gfCNCPoint1[20427] = {X 387.5470, Y 13.9480, Z -2.1667, A 0.000, B 0.000, C 0.000 }
gfCNCPoint1[20428] = {X 387.4498, Y 13.0232, Z -2.1667, A 0.000, B 0.000, C 0.000 }
gfCNCPoint1[20429] = {X 387.4496, Y 12.1868, Z -2.1667, A 0.000, B 0.000, C 0.000 }
gfCNCPoint1[20430] = {X 387.5362, Y 11.2718, Z -2.1667, A 0.000, B 0.000, C 0.000 }
gfCNCPoint1[20431] = {X 387.7928, Y 10.3892, Z -2.1667, A 0.000, B 0.000, C 0.000 }
gfCNCPoint1[20432] = {X 388.2375, Y 9.5281, Z -2.1667, A 0.000, B 0.000, C 0.000 }
gfCNCPoint1[20433] = {X 388.8436, Y 8.7718, Z -2.1667, A 0.000, B 0.000, C 0.000 }
gfCNCPoint1[20434] = {X 389.5872, Y 8.1503, Z -2.1667, A 0.000, B 0.000, C 0.000 }
gfCNCPoint1[20435] = {X 390.4390, Y 7.6880, Z -2.1667, A 0.000, B 0.000, C 0.000 }
gfCNCPoint1[20436] = {X 391.3653, Y 7.4030, Z -2.1667, A 0.000, B 0.000, C 0.000 }
gfCNCPoint1[20437] = {X 392.3296, Y 7.3068, Z -2.1667, A 0.000, B 0.000, C 0.000 }
gfCNCPoint1[20438] = {X 399.1118, Y 7.3068, Z -2.1667, A 0.000, B 0.000, C 0.000 }
gfCNCPoint1[20439] = {X 400.0638, Y 7.4006, Z -2.1667, A 0.000, B 0.000, C 0.000 }
gfCNCPoint1[20440] = {X 400.9793, Y 7.6783, Z -2.1667, A 0.000, B 0.000, C 0.000 }
gfCNCPoint1[20441] = {X 401.8229, Y 8.1292, Z -2.1667, A 0.000, B 0.000, C 0.000 }
gfCNCPoint1[20442] = {X 402.5624, Y 8.7361, Z -2.1667, A 0.000, B 0.000, C 0.000 }
gfCNCPoint1[20443] = {X 403.1693, Y 9.4756, Z -2.1667, A 0.000, B 0.000, C 0.000 }
gfCNCPoint1[20444] = {X 403.6203, Y 10.3193, Z -2.1667, A 0.000, B 0.000, C 0.000 }
gfCNCPoint1[20445] = {X 403.8980, Y 11.2348, Z -2.1667, A 0.000, B 0.000, C 0.000 }
gfCNCPoint1[20446] = {X 403.9918, Y 12.1868, Z -2.1667, A 0.000, B 0.000, C 0.000 }
gfCNCPoint1[20447] = {X 403.9915, Y 13.0237, Z -2.1667, A 0.000, B 0.000, C 0.000 }
gfCNCPoint1[20448] = {X 403.9016, Y 13.9115, Z -2.1667, A 0.000, B 0.000, C 0.000 }
gfCNCPoint1[20449] = {X 403.6516, Y 14.7680, Z -2.1667, A 0.000, B 0.000, C 0.000 }
gfCNCPoint1[20450] = {X 405.3653, Y 17.7437, Z -2.1667, A 0.000, B 0.000, C 0.000 }
gfCNCPoint1[20451] = {X 407.2450, Y 14.6988, Z -2.1667, A 0.000, B 0.000, C 0.000 }
gfCNCPoint1[20452] = {X 407.0143, Y 13.8732, Z -2.1667, A 0.000, B 0.000, C 0.000 }
gfCNCPoint1[20453] = {X 406.9317, Y 13.0199, Z -2.1667, A 0.000, B 0.000, C 0.000 }
gfCNCPoint1[20454] = {X 406.9315, Y 12.1868, Z -2.1667, A 0.000, B 0.000, C 0.000 }
gfCNCPoint1[20455] = {X 407.0253, Y 11.2348, Z -2.1667, A 0.000, B 0.000, C 0.000 }
gfCNCPoint1[20456] = {X 407.3030, Y 10.3193, Z -2.1667, A 0.000, B 0.000, C 0.000 }
gfCNCPoint1[20457] = {X 407.7540, Y 9.4756, Z -2.1667, A 0.000, B 0.000, C 0.000 }
gfCNCPoint1[20458] = {X 408.3609, Y 8.7361, Z -2.1667, A 0.000, B 0.000, C 0.000 }
gfCNCPoint1[20459] = {X 409.1004, Y 8.1292, Z -2.1667, A 0.000, B 0.000, C 0.000 }
gfCNCPoint1[20460] = {X 409.9440, Y 7.6783, Z -2.1667, A 0.000, B 0.000, C 0.000 }
gfCNCPoint1[20461] = {X 410.8595, Y 7.4006, Z -2.1667, A 0.000, B 0.000, C 0.000 }
gfCNCPoint1[20462] = {X 411.8115, Y 7.3068, Z -2.1667, A 0.000, B 0.000, C 0.000 }
gfCNCPoint1[20463] = {X 419.3245, Y 7.3068, Z -2.1667, A 0.000, B 0.000, C 0.000 }
gfCNCPoint1[20464] = {X 420.2888, Y 7.4030, Z -2.1667, A 0.000, B 0.000, C 0.000 }
gfCNCPoint1[20465] = {X 421.2151, Y 7.6880, Z -2.1667, A 0.000, B 0.000, C 0.000 }
gfCNCPoint1[20466] = {X 422.0669, Y 8.1503, Z -2.1667, A 0.000, B 0.000, C 0.000 }
gfCNCPoint1[20467] = {X 422.8105, Y 8.7718, Z -2.1667, A 0.000, B 0.000, C 0.000 }
gfCNCPoint1[20468] = {X 423.4166, Y 9.5281, Z -2.1667, A 0.000, B 0.000, C 0.000 }
gfCNCPoint1[20469] = {X 423.8613, Y 10.3892, Z -2.1667, A 0.000, B 0.000, C 0.000 }
gfCNCPoint1[20470] = {X 424.1179, Y 11.2718, Z -2.1667, A 0.000, B 0.000, C 0.000 }
gfCNCPoint1[20471] = {X 424.2045, Y 12.1868, Z -2.1667, A 0.000, B 0.000, C 0.000 }
gfCNCPoint1[20472] = {X 424.2045, Y 12.9779, Z -2.1667, A 0.000, B 0.000, C 0.000 }
gfCNCPoint1[20473] = {X 424.1055, Y 13.9307, Z -2.1667, A 0.000, B 0.000, C 0.000 }
gfCNCPoint1[20474] = {X 423.8248, Y 14.8465, Z -2.1667, A 0.000, B 0.000, C 0.000 }
gfCNCPoint1[20475] = {X 423.3729, Y 15.6910, Z -2.1667, A 0.000, B 0.000, C 0.000 }
gfCNCPoint1[20476] = {X 422.7668, Y 16.4327, Z -2.1667, A 0.000, B 0.000, C 0.000 }
gfCNCPoint1[20477] = {X 422.0290, Y 17.0436, Z -2.1667, A 0.000, B 0.000, C 0.000 }
gfCNCPoint1[20478] = {X 421.1874, Y 17.5009, Z -2.1667, A 0.000, B 0.000, C 0.000 }
gfCNCPoint1[20479] = {X 420.5395, Y 18.3844, Z -2.1667, A 0.000, B 0.000, C 0.000 }
gfCNCPoint1[20480] = {X 419.9503, Y 19.3080, Z -2.1667, A 0.000, B 0.000, C 0.000 }
gfCNCPoint1[20481] = {X 414.1631, Y 28.6162, Z -2.1667, A 0.000, B 0.000, C 0.000 }
gfCNCPoint1[20482] = {X 422.3159, Y 33.6850, Z -2.1667, A 0.000, B 0.000, C 0.000 }
gfCNCPoint1[20483] = {X 421.8891, Y 34.3715, Z -2.1667, A 0.000, B 0.000, C 0.000 }
gfCNCPoint1[20484] = {X 422.1457, Y 34.1014, Z -2.1667, A 0.000, B 0.000, C 0.000 }
gfCNCPoint1[20485] = {X 422.4091, Y 33.8380, Z -2.1667, A 0.000, B 0.000, C 0.000 }
gfCNCPoint1[20486] = {X 422.3623, Y 33.7616, Z -2.1667, A 0.000, B 0.000, C 0.000 }
gfCNCPoint1[20487] = {X 422.3159, Y 33.6850, Z -2.1667, A 0.000, B 0.000, C 0.000 }
gfCNCPoint1[20488] = {X 420.2777, Y 32.4178, Z -2.1667, A 0.000, B 0.000, C 0.000 }
gfCNCPoint1[20489] = {X 419.3062, Y 33.9804, Z -2.1667, A 0.000, B 0.000, C 0.000 }
gfCNCPoint1[20490] = {X 419.3065, Y 38.3391, Z -2.1667, A 0.000, B 0.000, C 0.000 }
gfCNCPoint1[20491] = {X 419.9570, Y 39.7077, Z -2.1667, A 0.000, B 0.000, C 0.000 }
gfCNCPoint1[20492] = {X 420.4329, Y 41.1464, Z -2.1667, A 0.000, B 0.000, C 0.000 }
gfCNCPoint1[20493] = {X 420.6276, Y 41.1585, Z -2.1667, A 0.000, B 0.000, C 0.000 }
gfCNCPoint1[20494] = {X 420.8222, Y 41.1728, Z -2.1667, A 0.000, B 0.000, C 0.000 }
gfCNCPoint1[20495] = {X 421.2839, Y 39.7588, Z -2.1667, A 0.000, B 0.000, C 0.000 }
gfCNCPoint1[20496] = {X 421.9160, Y 38.4123, Z -2.1667, A 0.000, B 0.000, C 0.000 }
gfCNCPoint1[20497] = {X 422.7087, Y 37.1536, Z -2.1667, A 0.000, B 0.000, C 0.000 }
gfCNCPoint1[20498] = {X 423.6502, Y 36.0020, Z -2.1667, A 0.000, B 0.000, C 0.000 }
gfCNCPoint1[20499] = {X 424.3400, Y 35.3147, Z -2.1667, A 0.000, B 0.000, C 0.000 }
gfCNCPoint1[20500] = {X 425.0829, Y 34.6852, Z -2.1667, A 0.000, B 0.000, C 0.000 }
gfCNCPoint1[20501] = {X 425.4264, Y 34.0128, Z -2.1667, A 0.000, B 0.000, C 0.000 }
gfCNCPoint1[20502] = {X 424.8791, Y 33.2419, Z -2.1667, A 0.000, B 0.000, C 0.000 }
gfCNCPoint1[20503] = {X 424.3706, Y 32.4448, Z -2.1667, A 0.000, B 0.000, C 0.000 }
gfCNCPoint1[20504] = {X 423.3899, Y 30.5981, Z -2.1667, A 0.000, B 0.000, C 0.000 }
gfCNCPoint1[20505] = {X 422.6170, Y 28.6551, Z -2.1667, A 0.000, B 0.000, C 0.000 }
gfCNCPoint1[20506] = {X 420.2777, Y 32.4178, Z -2.1667, A 0.000, B 0.000, C 0.000 }
gfCNCPoint1[20507] = {X 418.2395, Y 31.1506, Z -2.1667, A 0.000, B 0.000, C 0.000 }
gfCNCPoint1[20508] = {X 416.9061, Y 33.2953, Z -2.1667, A 0.000, B 0.000, C 0.000 }
gfCNCPoint1[20509] = {X 416.9065, Y 38.9959, Z -2.1667, A 0.000, B 0.000, C 0.000 }
gfCNCPoint1[20510] = {X 417.4880, Y 40.0490, Z -2.1667, A 0.000, B 0.000, C 0.000 }
gfCNCPoint1[20511] = {X 417.9361, Y 41.1653, Z -2.1667, A 0.000, B 0.000, C 0.000 }
gfCNCPoint1[20512] = {X 418.2441, Y 42.3282, Z -2.1667, A 0.000, B 0.000, C 0.000 }
gfCNCPoint1[20513] = {X 418.4074, Y 43.5200, Z -2.1667, A 0.000, B 0.000, C 0.000 }
gfCNCPoint1[20514] = {X 419.4886, Y 43.5200, Z -2.1667, A 0.000, B 0.000, C 0.000 }
gfCNCPoint1[20515] = {X 421.1752, Y 43.6186, Z -2.1667, A 0.000, B 0.000, C 0.000 }
gfCNCPoint1[20516] = {X 422.8389, Y 43.9129, Z -2.1667, A 0.000, B 0.000, C 0.000 }
gfCNCPoint1[20517] = {X 423.0005, Y 42.4234, Z -2.1667, A 0.000, B 0.000, C 0.000 }
gfCNCPoint1[20518] = {X 423.3900, Y 40.9766, Z -2.1667, A 0.000, B 0.000, C 0.000 }
gfCNCPoint1[20519] = {X 423.9980, Y 39.6073, Z -2.1667, A 0.000, B 0.000, C 0.000 }
gfCNCPoint1[20520] = {X 424.8102, Y 38.3482, Z -2.1667, A 0.000, B 0.000, C 0.000 }
gfCNCPoint1[20521] = {X 425.8068, Y 37.2295, Z -2.1667, A 0.000, B 0.000, C 0.000 }
gfCNCPoint1[20522] = {X 426.9642, Y 36.2780, Z -2.1667, A 0.000, B 0.000, C 0.000 }
gfCNCPoint1[20523] = {X 428.2766, Y 33.7091, Z -2.1667, A 0.000, B 0.000, C 0.000 }
gfCNCPoint1[20524] = {X 427.2128, Y 32.3915, Z -2.1667, A 0.000, B 0.000, C 0.000 }
gfCNCPoint1[20525] = {X 426.2880, Y 30.9728, Z -2.1667, A 0.000, B 0.000, C 0.000 }
gfCNCPoint1[20526] = {X 425.5119, Y 29.4677, Z -2.1667, A 0.000, B 0.000, C 0.000 }
gfCNCPoint1[20527] = {X 424.8924, Y 27.8916, Z -2.1667, A 0.000, B 0.000, C 0.000 }
gfCNCPoint1[20528] = {X 424.8106, Y 27.6414, Z -2.1667, A 0.000, B 0.000, C 0.000 }
gfCNCPoint1[20529] = {X 424.7328, Y 27.3900, Z -2.1667, A 0.000, B 0.000, C 0.000 }
gfCNCPoint1[20530] = {X 424.3001, Y 25.6524, Z -2.1667, A 0.000, B 0.000, C 0.000 }
gfCNCPoint1[20531] = {X 424.0106, Y 23.8853, Z -2.1667, A 0.000, B 0.000, C 0.000 }
gfCNCPoint1[20532] = {X 423.8662, Y 22.1005, Z -2.1667, A 0.000, B 0.000, C 0.000 }
gfCNCPoint1[20533] = {X 418.2395, Y 31.1506, Z -2.1667, A 0.000, B 0.000, C 0.000 }
gfCNCPoint1[20534] = {X 416.2013, Y 29.8834, Z -2.1667, A 0.000, B 0.000, C 0.000 }
gfCNCPoint1[20535] = {X 414.5060, Y 32.6101, Z -2.1667, A 0.000, B 0.000, C 0.000 }
gfCNCPoint1[20536] = {X 414.5066, Y 39.7473, Z -2.1667, A 0.000, B 0.000, C 0.000 }
gfCNCPoint1[20537] = {X 415.1552, Y 40.7521, Z -2.1667, A 0.000, B 0.000, C 0.000 }
gfCNCPoint1[20538] = {X 415.6336, Y 41.8482, Z -2.1667, A 0.000, B 0.000, C 0.000 }
gfCNCPoint1[20539] = {X 415.9293, Y 43.0070, Z -2.1667, A 0.000, B 0.000, C 0.000 }
gfCNCPoint1[20540] = {X 416.0347, Y 44.1983, Z -2.1667, A 0.000, B 0.000, C 0.000 }
gfCNCPoint1[20541] = {X 416.0347, Y 44.9999, Z -2.1667, A 0.000, B 0.000, C 0.000 }
gfCNCPoint1[20542] = {X 416.0201, Y 45.4609, Z -2.1667, A 0.000, B 0.000, C 0.000 }
gfCNCPoint1[20543] = {X 415.9763, Y 45.9200, Z -2.1667, A 0.000, B 0.000, C 0.000 }
gfCNCPoint1[20544] = {X 419.4886, Y 45.9200, Z -2.1667, A 0.000, B 0.000, C 0.000 }
gfCNCPoint1[20545] = {X 420.8957, Y 46.0022, Z -2.1667, A 0.000, B 0.000, C 0.000 }
gfCNCPoint1[20546] = {X 422.2836, Y 46.2478, Z -2.1667, A 0.000, B 0.000, C 0.000 }
gfCNCPoint1[20547] = {X 423.4822, Y 46.5992, Z -2.1667, A 0.000, B 0.000, C 0.000 }
gfCNCPoint1[20548] = {X 424.6380, Y 47.0725, Z -2.1667, A 0.000, B 0.000, C 0.000 }
gfCNCPoint1[20549] = {X 425.7388, Y 47.6626, Z -2.1667, A 0.000, B 0.000, C 0.000 }
gfCNCPoint1[20550] = {X 425.4600, Y 46.7984, Z -2.1667, A 0.000, B 0.000, C 0.000 }
gfCNCPoint1[20551] = {X 425.2910, Y 45.9063, Z -2.1667, A 0.000, B 0.000, C 0.000 }
gfCNCPoint1[20552] = {X 425.2344, Y 45.0000, Z -2.1667, A 0.000, B 0.000, C 0.000 }
gfCNCPoint1[20553] = {X 425.2344, Y 44.2090, Z -2.1667, A 0.000, B 0.000, C 0.000 }
gfCNCPoint1[20554] = {X 425.2353, Y 44.0976, Z -2.1667, A 0.000, B 0.000, C 0.000 }
gfCNCPoint1[20555] = {X 425.2378, Y 43.9863, Z -2.1667, A 0.000, B 0.000, C 0.000 }
gfCNCPoint1[20556] = {X 425.3770, Y 42.7748, Z -2.1667, A 0.000, B 0.000, C 0.000 }
gfCNCPoint1[20557] = {X 425.7165, Y 41.6036, Z -2.1667, A 0.000, B 0.000, C 0.000 }
gfCNCPoint1[20558] = {X 426.2468, Y 40.5054, Z -2.1667, A 0.000, B 0.000, C 0.000 }
gfCNCPoint1[20559] = {X 426.9528, Y 39.5112, Z -2.1667, A 0.000, B 0.000, C 0.000 }
gfCNCPoint1[20560] = {X 427.8150, Y 38.6488, Z -2.1667, A 0.000, B 0.000, C 0.000 }
gfCNCPoint1[20561] = {X 428.8090, Y 37.9424, Z -2.1667, A 0.000, B 0.000, C 0.000 }
gfCNCPoint1[20562] = {X 431.2071, Y 33.2482, Z -2.1667, A 0.000, B 0.000, C 0.000 }
gfCNCPoint1[20563] = {X 430.0935, Y 32.1404, Z -2.1667, A 0.000, B 0.000, C 0.000 }
gfCNCPoint1[20564] = {X 429.1082, Y 30.9169, Z -2.1667, A 0.000, B 0.000, C 0.000 }
gfCNCPoint1[20565] = {X 428.2633, Y 29.5927, Z -2.1667, A 0.000, B 0.000, C 0.000 }
gfCNCPoint1[20566] = {X 427.5689, Y 28.1837, Z -2.1667, A 0.000, B 0.000, C 0.000 }
gfCNCPoint1[20567] = {X 427.0335, Y 26.7069, Z -2.1667, A 0.000, B 0.000, C 0.000 }
gfCNCPoint1[20568] = {X 426.6495, Y 25.1622, Z -2.1667, A 0.000, B 0.000, C 0.000 }
gfCNCPoint1[20569] = {X 426.3925, Y 23.5913, Z -2.1667, A 0.000, B 0.000, C 0.000 }
gfCNCPoint1[20570] = {X 426.2643, Y 22.0048, Z -2.1667, A 0.000, B 0.000, C 0.000 }
gfCNCPoint1[20571] = {X 426.2911, Y 19.9392, Z -2.1667, A 0.000, B 0.000, C 0.000 }
gfCNCPoint1[20572] = {X 426.5359, Y 17.8880, Z -2.1667, A 0.000, B 0.000, C 0.000 }
gfCNCPoint1[20573] = {X 426.9959, Y 15.8741, Z -2.1667, A 0.000, B 0.000, C 0.000 }
gfCNCPoint1[20574] = {X 427.6134, Y 14.1183, Z -2.1667, A 0.000, B 0.000, C 0.000 }
gfCNCPoint1[20575] = {X 428.4471, Y 12.4541, Z -2.1667, A 0.000, B 0.000, C 0.000 }
gfCNCPoint1[20576] = {X 429.4837, Y 10.9082, Z -2.1667, A 0.000, B 0.000, C 0.000 }
gfCNCPoint1[20577] = {X 430.7066, Y 9.5051, Z -2.1667, A 0.000, B 0.000, C 0.000 }
gfCNCPoint1[20578] = {X 426.0925, Y 9.5051, Z -2.1667, A 0.000, B 0.000, C 0.000 }
gfCNCPoint1[20579] = {X 426.3754, Y 10.3751, Z -2.1667, A 0.000, B 0.000, C 0.000 }
gfCNCPoint1[20580] = {X 426.5470, Y 11.2738, Z -2.1667, A 0.000, B 0.000, C 0.000 }
gfCNCPoint1[20581] = {X 426.6045, Y 12.1868, Z -2.1667, A 0.000, B 0.000, C 0.000 }
gfCNCPoint1[20582] = {X 426.6045, Y 12.9858, Z -2.1667, A 0.000, B 0.000, C 0.000 }
gfCNCPoint1[20583] = {X 426.4810, Y 14.2875, Z -2.1667, A 0.000, B 0.000, C 0.000 }
gfCNCPoint1[20584] = {X 426.1288, Y 15.5467, Z -2.1667, A 0.000, B 0.000, C 0.000 }
gfCNCPoint1[20585] = {X 425.5589, Y 16.7235, Z -2.1667, A 0.000, B 0.000, C 0.000 }
gfCNCPoint1[20586] = {X 424.7895, Y 17.7807, Z -2.1667, A 0.000, B 0.000, C 0.000 }
gfCNCPoint1[20587] = {X 423.8449, Y 18.6847, Z -2.1667, A 0.000, B 0.000, C 0.000 }
gfCNCPoint1[20588] = {X 422.7549, Y 19.4070, Z -2.1667, A 0.000, B 0.000, C 0.000 }
gfCNCPoint1[20589] = {X 422.3647, Y 19.9716, Z -2.1667, A 0.000, B 0.000, C 0.000 }
gfCNCPoint1[20590] = {X 422.0017, Y 20.5540, Z -2.1667, A 0.000, B 0.000, C 0.000 }
gfCNCPoint1[20591] = {X 416.2013, Y 29.8834, Z -2.1667, A 0.000, B 0.000, C 0.000 }
gfCNCPoint1[20592] = {X 414.1631, Y 28.6162, Z -2.1667, A 0.000, B 0.000, C 0.000 }
gfCNCPoint1[20593] = {X 412.1060, Y 31.9249, Z -2.1667, A 0.000, B 0.000, C 0.000 }
gfCNCPoint1[20594] = {X 412.1067, Y 40.6523, Z -2.1667, A 0.000, B 0.000, C 0.000 }
gfCNCPoint1[20595] = {X 412.7484, Y 41.4088, Z -2.1667, A 0.000, B 0.000, C 0.000 }
gfCNCPoint1[20596] = {X 413.2283, Y 42.2769, Z -2.1667, A 0.000, B 0.000, C 0.000 }
gfCNCPoint1[20597] = {X 413.5277, Y 43.2227, Z -2.1667, A 0.000, B 0.000, C 0.000 }
gfCNCPoint1[20598] = {X 413.6347, Y 44.2089, Z -2.1667, A 0.000, B 0.000, C 0.000 }
gfCNCPoint1[20599] = {X 413.6347, Y 45.0000, Z -2.1667, A 0.000, B 0.000, C 0.000 }
gfCNCPoint1[20600] = {X 413.6249, Y 45.3090, Z -2.1667, A 0.000, B 0.000, C 0.000 }
gfCNCPoint1[20601] = {X 413.5956, Y 45.6167, Z -2.1667, A 0.000, B 0.000, C 0.000 }
gfCNCPoint1[20602] = {X 413.3652, Y 46.5992, Z -2.1667, A 0.000, B 0.000, C 0.000 }
gfCNCPoint1[20603] = {X 412.9377, Y 47.5134, Z -2.1667, A 0.000, B 0.000, C 0.000 }
gfCNCPoint1[20604] = {X 412.3313, Y 48.3200, Z -2.1667, A 0.000, B 0.000, C 0.000 }
gfCNCPoint1[20605] = {X 411.9795, Y 47.9934, Z -2.1667, A 0.000, B 0.000, C 0.000 }
gfCNCPoint1[20606] = {X 411.3003, Y 48.5889, Z -2.1667, A 0.000, B 0.000, C 0.000 }
gfCNCPoint1[20607] = {X 410.5138, Y 49.0331, Z -2.1667, A 0.000, B 0.000, C 0.000 }
gfCNCPoint1[20608] = {X 409.6532, Y 49.3073, Z -2.1667, A 0.000, B 0.000, C 0.000 }
gfCNCPoint1[20609] = {X 408.7547, Y 49.4000, Z -2.1667, A 0.000, B 0.000, C 0.000 }
gfCNCPoint1[20610] = {X 402.3112, Y 49.4000, Z -2.1667, A 0.000, B 0.000, C 0.000 }
gfCNCPoint1[20611] = {X 401.3321, Y 49.2897, Z -2.1667, A 0.000, B 0.000, C 0.000 }
gfCNCPoint1[20612] = {X 400.4021, Y 48.9643, Z -2.1667, A 0.000, B 0.000, C 0.000 }
gfCNCPoint1[20613] = {X 399.5678, Y 48.4400, Z -2.1667, A 0.000, B 0.000, C 0.000 }
gfCNCPoint1[20614] = {X 398.8711, Y 47.7433, Z -2.1667, A 0.000, B 0.000, C 0.000 }
gfCNCPoint1[20615] = {X 398.3469, Y 46.9091, Z -2.1667, A 0.000, B 0.000, C 0.000 }
gfCNCPoint1[20616] = {X 398.0215, Y 45.9791, Z -2.1667, A 0.000, B 0.000, C 0.000 }
gfCNCPoint1[20617] = {X 397.9112, Y 45.0000, Z -2.1667, A 0.000, B 0.000, C 0.000 }
gfCNCPoint1[20618] = {X 397.9116, Y 44.1518, Z -2.1667, A 0.000, B 0.000, C 0.000 }
gfCNCPoint1[20619] = {X 398.0215, Y 43.2300, Z -2.1667, A 0.000, B 0.000, C 0.000 }
gfCNCPoint1[20620] = {X 398.3223, Y 42.3519, Z -2.1667, A 0.000, B 0.000, C 0.000 }
gfCNCPoint1[20621] = {X 398.8006, Y 41.5563, Z -2.1667, A 0.000, B 0.000, C 0.000 }
gfCNCPoint1[20622] = {X 399.4352, Y 40.8789, Z -2.1667, A 0.000, B 0.000, C 0.000 }
gfCNCPoint1[20623] = {X 399.4352, Y 31.6934, Z -2.1667, A 0.000, B 0.000, C 0.000 }
gfCNCPoint1[20624] = {X 393.2514, Y 20.9402, Z -2.1667, A 0.000, B 0.000, C 0.000 }
gfCNCPoint1[20625] = {X 392.4348, Y 19.5574, Z -2.1667, A 0.000, B 0.000, C 0.000 }
gfCNCPoint1[20626] = {X 391.5867, Y 18.1938, Z -2.1667, A 0.000, B 0.000, C 0.000 }
gfCNCPoint1[20627] = {X 391.1415, Y 17.5837, Z -2.1667, A 0.000, B 0.000, C 0.000 }
gfCNCPoint1[20628] = {X 390.6238, Y 17.0339, Z -2.1667, A 0.000, B 0.000, C 0.000 }
gfCNCPoint1[20629] = {X 389.8686, Y 16.6254, Z -2.1667, A 0.000, B 0.000, C 0.000 }
gfCNCPoint1[20630] = {X 389.2071, Y 16.0780, Z -2.1667, A 0.000, B 0.000, C 0.000 }
gfCNCPoint1[20631] = {X 388.6645, Y 15.4125, Z -2.1667, A 0.000, B 0.000, C 0.000 }
gfCNCPoint1[20632] = {X 388.2615, Y 14.6544, Z -2.1667, A 0.000, B 0.000, C 0.000 }
gfCNCPoint1[20633] = {X 388.0134, Y 13.8324, Z -2.1667, A 0.000, B 0.000, C 0.000 }
gfCNCPoint1[20634] = {X 387.9296, Y 12.9779, Z -2.1667, A 0.000, B 0.000, C 0.000 }
gfCNCPoint1[20635] = {X 387.9296, Y 12.1868, Z -2.1667, A 0.000, B 0.000, C 0.000 }
gfCNCPoint1[20636] = {X 388.0399, Y 11.2077, Z -2.1667, A 0.000, B 0.000, C 0.000 }
gfCNCPoint1[20637] = {X 388.3654, Y 10.2777, Z -2.1667, A 0.000, B 0.000, C 0.000 }
gfCNCPoint1[20638] = {X 388.8896, Y 9.4435, Z -2.1667, A 0.000, B 0.000, C 0.000 }
gfCNCPoint1[20639] = {X 389.5863, Y 8.7468, Z -2.1667, A 0.000, B 0.000, C 0.000 }
gfCNCPoint1[20640] = {X 390.4205, Y 8.2226, Z -2.1667, A 0.000, B 0.000, C 0.000 }
gfCNCPoint1[20641] = {X 391.3505, Y 7.8971, Z -2.1667, A 0.000, B 0.000, C 0.000 }
gfCNCPoint1[20642] = {X 392.3296, Y 7.7868, Z -2.1667, A 0.000, B 0.000, C 0.000 }
gfCNCPoint1[20643] = {X 399.1118, Y 7.7868, Z -2.1667, A 0.000, B 0.000, C 0.000 }
gfCNCPoint1[20644] = {X 400.0909, Y 7.8971, Z -2.1667, A 0.000, B 0.000, C 0.000 }
gfCNCPoint1[20645] = {X 401.0208, Y 8.2226, Z -2.1667, A 0.000, B 0.000, C 0.000 }
gfCNCPoint1[20646] = {X 401.8551, Y 8.7468, Z -2.1667, A 0.000, B 0.000, C 0.000 }
gfCNCPoint1[20647] = {X 402.5518, Y 9.4435, Z -2.1667, A 0.000, B 0.000, C 0.000 }
gfCNCPoint1[20648] = {X 403.0760, Y 10.2777, Z -2.1667, A 0.000, B 0.000, C 0.000 }
gfCNCPoint1[20649] = {X 403.4014, Y 11.2077, Z -2.1667, A 0.000, B 0.000, C 0.000 }
gfCNCPoint1[20650] = {X 403.5118, Y 12.1868, Z -2.1667, A 0.000, B 0.000, C 0.000 }
gfCNCPoint1[20651] = {X 403.5115, Y 13.0233, Z -2.1667, A 0.000, B 0.000, C 0.000 }
gfCNCPoint1[20652] = {X 403.4070, Y 13.9326, Z -2.1667, A 0.000, B 0.000, C 0.000 }
gfCNCPoint1[20653] = {X 403.1165, Y 14.8007, Z -2.1667, A 0.000, B 0.000, C 0.000 }
gfCNCPoint1[20654] = {X 405.3510, Y 18.6806, Z -2.1667, A 0.000, B 0.000, C 0.000 }
gfCNCPoint1[20655] = {X 407.7814, Y 14.7438, Z -2.1667, A 0.000, B 0.000, C 0.000 }
gfCNCPoint1[20656] = {X 407.5050, Y 13.8800, Z -2.1667, A 0.000, B 0.000, C 0.000 }
gfCNCPoint1[20657] = {X 407.4115, Y 12.9779, Z -2.1667, A 0.000, B 0.000, C 0.000 }
gfCNCPoint1[20658] = {X 407.4115, Y 12.1868, Z -2.1667, A 0.000, B 0.000, C 0.000 }
gfCNCPoint1[20659] = {X 407.5219, Y 11.2077, Z -2.1667, A 0.000, B 0.000, C 0.000 }
gfCNCPoint1[20660] = {X 407.8473, Y 10.2777, Z -2.1667, A 0.000, B 0.000, C 0.000 }
gfCNCPoint1[20661] = {X 408.3715, Y 9.4435, Z -2.1667, A 0.000, B 0.000, C 0.000 }
gfCNCPoint1[20662] = {X 409.0682, Y 8.7468, Z -2.1667, A 0.000, B 0.000, C 0.000 }
gfCNCPoint1[20663] = {X 409.9024, Y 8.2226, Z -2.1667, A 0.000, B 0.000, C 0.000 }
gfCNCPoint1[20664] = {X 410.8324, Y 7.8971, Z -2.1667, A 0.000, B 0.000, C 0.000 }
gfCNCPoint1[20665] = {X 411.8115, Y 7.7868, Z -2.1667, A 0.000, B 0.000, C 0.000 }
gfCNCPoint1[20666] = {X 419.3245, Y 7.7868, Z -2.1667, A 0.000, B 0.000, C 0.000 }
gfCNCPoint1[20667] = {X 420.3036, Y 7.8971, Z -2.1667, A 0.000, B 0.000, C 0.000 }
gfCNCPoint1[20668] = {X 421.2335, Y 8.2226, Z -2.1667, A 0.000, B 0.000, C 0.000 }
gfCNCPoint1[20669] = {X 422.0678, Y 8.7468, Z -2.1667, A 0.000, B 0.000, C 0.000 }
gfCNCPoint1[20670] = {X 422.7645, Y 9.4435, Z -2.1667, A 0.000, B 0.000, C 0.000 }
gfCNCPoint1[20671] = {X 423.2887, Y 10.2777, Z -2.1667, A 0.000, B 0.000, C 0.000 }
gfCNCPoint1[20672] = {X 423.6141, Y 11.2077, Z -2.1667, A 0.000, B 0.000, C 0.000 }
gfCNCPoint1[20673] = {X 423.7245, Y 12.1868, Z -2.1667, A 0.000, B 0.000, C 0.000 }
gfCNCPoint1[20674] = {X 423.7244, Y 12.9811, Z -2.1667, A 0.000, B 0.000, C 0.000 }
gfCNCPoint1[20675] = {X 423.6301, Y 13.8598, Z -2.1667, A 0.000, B 0.000, C 0.000 }
gfCNCPoint1[20676] = {X 423.3645, Y 14.7028, Z -2.1667, A 0.000, B 0.000, C 0.000 }
gfCNCPoint1[20677] = {X 422.9382, Y 15.4769, Z -2.1667, A 0.000, B 0.000, C 0.000 }
gfCNCPoint1[20678] = {X 422.3679, Y 16.1520, Z -2.1667, A 0.000, B 0.000, C 0.000 }
gfCNCPoint1[20679] = {X 421.6758, Y 16.7016, Z -2.1667, A 0.000, B 0.000, C 0.000 }
gfCNCPoint1[20680] = {X 420.8891, Y 17.1042, Z -2.1667, A 0.000, B 0.000, C 0.000 }
gfCNCPoint1[20681] = {X 420.1821, Y 18.0570, Z -2.1667, A 0.000, B 0.000, C 0.000 }
gfCNCPoint1[20682] = {X 419.5419, Y 19.0558, Z -2.1667, A 0.000, B 0.000, C 0.000 }
gfCNCPoint1[20683] = {X 418.0618, Y 21.4528, Z -2.1667, A 0.000, B 0.000, C 0.000 }
gfCNCPoint1[20684] = {X 411.6260, Y 31.7877, Z -2.1667, A 0.000, B 0.000, C 0.000 }
gfCNCPoint1[20685] = {X 411.6267, Y 40.8621, Z -2.1667, A 0.000, B 0.000, C 0.000 }
gfCNCPoint1[20686] = {X 412.2657, Y 41.5589, Z -2.1667, A 0.000, B 0.000, C 0.000 }
gfCNCPoint1[20687] = {X 412.7461, Y 42.3733, Z -2.1667, A 0.000, B 0.000, C 0.000 }
gfCNCPoint1[20688] = {X 413.0467, Y 43.2696, Z -2.1667, A 0.000, B 0.000, C 0.000 }
gfCNCPoint1[20689] = {X 413.1547, Y 44.2089, Z -2.1667, A 0.000, B 0.000, C 0.000 }
gfCNCPoint1[20690] = {X 413.1545, Y 45.0423, Z -2.1667, A 0.000, B 0.000, C 0.000 }
gfCNCPoint1[20691] = {X 413.0719, Y 45.8494, Z -2.1667, A 0.000, B 0.000, C 0.000 }
gfCNCPoint1[20692] = {X 412.8426, Y 46.6276, Z -2.1667, A 0.000, B 0.000, C 0.000 }
gfCNCPoint1[20693] = {X 412.4743, Y 47.3505, Z -2.1667, A 0.000, B 0.000, C 0.000 }
gfCNCPoint1[20694] = {X 411.9795, Y 47.9934, Z -2.1667, A 0.000, B 0.000, C 0.000 }
gfCNCPoint1[20695] = {X 412.3313, Y 48.3200, Z -2.1667, A 0.000, B 0.000, C 0.000 }
gfCNCPoint1[20696] = {X 419.4886, Y 48.3200, Z -2.1667, A 0.000, B 0.000, C 0.000 }
gfCNCPoint1[20697] = {X 420.8006, Y 48.4093, Z -2.1667, A 0.000, B 0.000, C 0.000 }
gfCNCPoint1[20698] = {X 422.0883, Y 48.6756, Z -2.1667, A 0.000, B 0.000, C 0.000 }
gfCNCPoint1[20699] = {X 423.3281, Y 49.1140, Z -2.1667, A 0.000, B 0.000, C 0.000 }
gfCNCPoint1[20700] = {X 424.4970, Y 49.7164, Z -2.1667, A 0.000, B 0.000, C 0.000 }
gfCNCPoint1[20701] = {X 425.4625, Y 50.3832, Z -2.1667, A 0.000, B 0.000, C 0.000 }
gfCNCPoint1[20702] = {X 426.3402, Y 51.1620, Z -2.1667, A 0.000, B 0.000, C 0.000 }
gfCNCPoint1[20703] = {X 427.1172, Y 52.0412, Z -2.1667, A 0.000, B 0.000, C 0.000 }
gfCNCPoint1[20704] = {X 427.7821, Y 53.0080, Z -2.1667, A 0.000, B 0.000, C 0.000 }
gfCNCPoint1[20705] = {X 428.1269, Y 53.6317, Z -2.1667, A 0.000, B 0.000, C 0.000 }
gfCNCPoint1[20706] = {X 428.4249, Y 54.2792, Z -2.1667, A 0.000, B 0.000, C 0.000 }
gfCNCPoint1[20707] = {X 431.5823, Y 55.5098, Z -2.1667, A 0.000, B 0.000, C 0.000 }
gfCNCPoint1[20708] = {X 439.8770, Y 58.8007, Z -2.1667, A 0.000, B 0.000, C 0.000 }
gfCNCPoint1[20709] = {X 441.6471, Y 54.3390, Z -2.1667, A 0.000, B 0.000, C 0.000 }
gfCNCPoint1[20710] = {X 444.2222, Y 55.3606, Z -2.1667, A 0.000, B 0.000, C 0.000 }
gfCNCPoint1[20711] = {X 444.5425, Y 54.0020, Z -2.1667, A 0.000, B 0.000, C 0.000 }
gfCNCPoint1[20712] = {X 444.9921, Y 52.6806, Z -2.1667, A 0.000, B 0.000, C 0.000 }
gfCNCPoint1[20713] = {X 443.9519, Y 53.3765, Z -2.1667, A 0.000, B 0.000, C 0.000 }
gfCNCPoint1[20714] = {X 442.8307, Y 53.9324, Z -2.1667, A 0.000, B 0.000, C 0.000 }
gfCNCPoint1[20715] = {X 441.6471, Y 54.3390, Z -2.1667, A 0.000, B 0.000, C 0.000 }
gfCNCPoint1[20716] = {X 440.7621, Y 56.5698, Z -2.1667, A 0.000, B 0.000, C 0.000 }
gfCNCPoint1[20717] = {X 446.3797, Y 58.7986, Z -2.1667, A 0.000, B 0.000, C 0.000 }
gfCNCPoint1[20718] = {X 446.3796, Y 58.0000, Z -2.1667, A 0.000, B 0.000, C 0.000 }
gfCNCPoint1[20719] = {X 446.4303, Y 56.8944, Z -2.1667, A 0.000, B 0.000, C 0.000 }
gfCNCPoint1[20720] = {X 446.5820, Y 55.7981, Z -2.1667, A 0.000, B 0.000, C 0.000 }
gfCNCPoint1[20721] = {X 446.8492, Y 54.6647, Z -2.1667, A 0.000, B 0.000, C 0.000 }
gfCNCPoint1[20722] = {X 447.2243, Y 53.5622, Z -2.1667, A 0.000, B 0.000, C 0.000 }
gfCNCPoint1[20723] = {X 447.8767, Y 52.1752, Z -2.1667, A 0.000, B 0.000, C 0.000 }
gfCNCPoint1[20724] = {X 448.6995, Y 50.8820, Z -2.1667, A 0.000, B 0.000, C 0.000 }
gfCNCPoint1[20725] = {X 447.8224, Y 50.1272, Z -2.1667, A 0.000, B 0.000, C 0.000 }
gfCNCPoint1[20726] = {X 447.0760, Y 49.2431, Z -2.1667, A 0.000, B 0.000, C 0.000 }
gfCNCPoint1[20727] = {X 446.4792, Y 48.2518, Z -2.1667, A 0.000, B 0.000, C 0.000 }
gfCNCPoint1[20728] = {X 446.0469, Y 47.1785, Z -2.1667, A 0.000, B 0.000, C 0.000 }
gfCNCPoint1[20729] = {X 445.6333, Y 48.2126, Z -2.1667, A 0.000, B 0.000, C 0.000 }
gfCNCPoint1[20730] = {X 445.0668, Y 49.1715, Z -2.1667, A 0.000, B 0.000, C 0.000 }
gfCNCPoint1[20731] = {X 444.3606, Y 50.0328, Z -2.1667, A 0.000, B 0.000, C 0.000 }
gfCNCPoint1[20732] = {X 443.5314, Y 50.7763, Z -2.1667, A 0.000, B 0.000, C 0.000 }
gfCNCPoint1[20733] = {X 442.7491, Y 51.2997, Z -2.1667, A 0.000, B 0.000, C 0.000 }
gfCNCPoint1[20734] = {X 441.9059, Y 51.7177, Z -2.1667, A 0.000, B 0.000, C 0.000 }
gfCNCPoint1[20735] = {X 441.0157, Y 52.0235, Z -2.1667, A 0.000, B 0.000, C 0.000 }
gfCNCPoint1[20736] = {X 440.0666, Y 52.2156, Z -2.1667, A 0.000, B 0.000, C 0.000 }
gfCNCPoint1[20737] = {X 439.1005, Y 52.2800, Z -2.1667, A 0.000, B 0.000, C 0.000 }
gfCNCPoint1[20738] = {X 432.5144, Y 52.2800, Z -2.1667, A 0.000, B 0.000, C 0.000 }
gfCNCPoint1[20739] = {X 431.6034, Y 52.2228, Z -2.1667, A 0.000, B 0.000, C 0.000 }
gfCNCPoint1[20740] = {X 430.7066, Y 52.0520, Z -2.1667, A 0.000, B 0.000, C 0.000 }
gfCNCPoint1[20741] = {X 429.8384, Y 51.7703, Z -2.1667, A 0.000, B 0.000, C 0.000 }
gfCNCPoint1[20742] = {X 430.0172, Y 52.0776, Z -2.1667, A 0.000, B 0.000, C 0.000 }
gfCNCPoint1[20743] = {X 430.1870, Y 52.3901, Z -2.1667, A 0.000, B 0.000, C 0.000 }
gfCNCPoint1[20744] = {X 432.4640, Y 53.2776, Z -2.1667, A 0.000, B 0.000, C 0.000 }
gfCNCPoint1[20745] = {X 440.7621, Y 56.5698, Z -2.1667, A 0.000, B 0.000, C 0.000 }
gfCNCPoint1[20746] = {X 439.8770, Y 58.8007, Z -2.1667, A 0.000, B 0.000, C 0.000 }
gfCNCPoint1[20747] = {X 449.5098, Y 62.6225, Z -2.1667, A 0.000, B 0.000, C 0.000 }
gfCNCPoint1[20748] = {X 449.1115, Y 61.4473, Z -2.1667, A 0.000, B 0.000, C 0.000 }
gfCNCPoint1[20749] = {X 448.8668, Y 60.2308, Z -2.1667, A 0.000, B 0.000, C 0.000 }
gfCNCPoint1[20750] = {X 448.7798, Y 58.9930, Z -2.1667, A 0.000, B 0.000, C 0.000 }
gfCNCPoint1[20751] = {X 448.7796, Y 58.0000, Z -2.1667, A 0.000, B 0.000, C 0.000 }
gfCNCPoint1[20752] = {X 448.8564, Y 56.7833, Z -2.1667, A 0.000, B 0.000, C 0.000 }
gfCNCPoint1[20753] = {X 449.0855, Y 55.5859, Z -2.1667, A 0.000, B 0.000, C 0.000 }
gfCNCPoint1[20754] = {X 449.4632, Y 54.4268, Z -2.1667, A 0.000, B 0.000, C 0.000 }
gfCNCPoint1[20755] = {X 449.9837, Y 53.3244, Z -2.1667, A 0.000, B 0.000, C 0.000 }
gfCNCPoint1[20756] = {X 450.6386, Y 52.2961, Z -2.1667, A 0.000, B 0.000, C 0.000 }
gfCNCPoint1[20757] = {X 451.3887, Y 51.3890, Z -2.1667, A 0.000, B 0.000, C 0.000 }
gfCNCPoint1[20758] = {X 452.2434, Y 50.5796, Z -2.1667, A 0.000, B 0.000, C 0.000 }
gfCNCPoint1[20759] = {X 453.1901, Y 49.8800, Z -2.1667, A 0.000, B 0.000, C 0.000 }
gfCNCPoint1[20760] = {X 452.3731, Y 49.8442, Z -2.1667, A 0.000, B 0.000, C 0.000 }
gfCNCPoint1[20761] = {X 451.5735, Y 49.6724, Z -2.1667, A 0.000, B 0.000, C 0.000 }
gfCNCPoint1[20762] = {X 450.8138, Y 49.3696, Z -2.1667, A 0.000, B 0.000, C 0.000 }
gfCNCPoint1[20763] = {X 450.1154, Y 48.9441, Z -2.1667, A 0.000, B 0.000, C 0.000 }
gfCNCPoint1[20764] = {X 449.3503, Y 48.2496, Z -2.1667, A 0.000, B 0.000, C 0.000 }
gfCNCPoint1[20765] = {X 448.7486, Y 47.4095, Z -2.1667, A 0.000, B 0.000, C 0.000 }
gfCNCPoint1[20766] = {X 448.3373, Y 46.4616, Z -2.1667, A 0.000, B 0.000, C 0.000 }
gfCNCPoint1[20767] = {X 448.1732, Y 45.7588, Z -2.1667, A 0.000, B 0.000, C 0.000 }
gfCNCPoint1[20768] = {X 448.1146, Y 45.0395, Z -2.1667, A 0.000, B 0.000, C 0.000 }
gfCNCPoint1[20769] = {X 448.1149, Y 44.1416, Z -2.1667, A 0.000, B 0.000, C 0.000 }
gfCNCPoint1[20770] = {X 448.2252, Y 43.1751, Z -2.1667, A 0.000, B 0.000, C 0.000 }
gfCNCPoint1[20771] = {X 448.5250, Y 42.2497, Z -2.1667, A 0.000, B 0.000, C 0.000 }
gfCNCPoint1[20772] = {X 449.0024, Y 41.4020, Z -2.1667, A 0.000, B 0.000, C 0.000 }
gfCNCPoint1[20773] = {X 449.6384, Y 40.6660, Z -2.1667, A 0.000, B 0.000, C 0.000 }
gfCNCPoint1[20774] = {X 449.6384, Y 35.0338, Z -2.1667, A 0.000, B 0.000, C 0.000 }
gfCNCPoint1[20775] = {X 447.8156, Y 35.0338, Z -2.1667, A 0.000, B 0.000, C 0.000 }
gfCNCPoint1[20776] = {X 443.7924, Y 42.8669, Z -2.1667, A 0.000, B 0.000, C 0.000 }
gfCNCPoint1[20777] = {X 443.9301, Y 43.5098, Z -2.1667, A 0.000, B 0.000, C 0.000 }
gfCNCPoint1[20778] = {X 443.9803, Y 44.1653, Z -2.1667, A 0.000, B 0.000, C 0.000 }
gfCNCPoint1[20779] = {X 443.9805, Y 45.0000, Z -2.1667, A 0.000, B 0.000, C 0.000 }
gfCNCPoint1[20780] = {X 443.9242, Y 45.7387, Z -2.1667, A 0.000, B 0.000, C 0.000 }
gfCNCPoint1[20781] = {X 443.7568, Y 46.4603, Z -2.1667, A 0.000, B 0.000, C 0.000 }
gfCNCPoint1[20782] = {X 443.3474, Y 47.4038, Z -2.1667, A 0.000, B 0.000, C 0.000 }
gfCNCPoint1[20783] = {X 442.7493, Y 48.2405, Z -2.1667, A 0.000, B 0.000, C 0.000 }
gfCNCPoint1[20784] = {X 441.9891, Y 48.9332, Z -2.1667, A 0.000, B 0.000, C 0.000 }
gfCNCPoint1[20785] = {X 441.1006, Y 49.4513, Z -2.1667, A 0.000, B 0.000, C 0.000 }
gfCNCPoint1[20786] = {X 440.1232, Y 49.7716, Z -2.1667, A 0.000, B 0.000, C 0.000 }
gfCNCPoint1[20787] = {X 439.1005, Y 49.8800, Z -2.1667, A 0.000, B 0.000, C 0.000 }
gfCNCPoint1[20788] = {X 432.5144, Y 49.8800, Z -2.1667, A 0.000, B 0.000, C 0.000 }
gfCNCPoint1[20789] = {X 431.6014, Y 49.7938, Z -2.1667, A 0.000, B 0.000, C 0.000 }
gfCNCPoint1[20790] = {X 430.7206, Y 49.5383, Z -2.1667, A 0.000, B 0.000, C 0.000 }
gfCNCPoint1[20791] = {X 429.8343, Y 49.0782, Z -2.1667, A 0.000, B 0.000, C 0.000 }
gfCNCPoint1[20792] = {X 429.0603, Y 48.4473, Z -2.1667, A 0.000, B 0.000, C 0.000 }
gfCNCPoint1[20793] = {X 428.4309, Y 47.6720, Z -2.1667, A 0.000, B 0.000, C 0.000 }
gfCNCPoint1[20794] = {X 427.9725, Y 46.7848, Z -2.1667, A 0.000, B 0.000, C 0.000 }
gfCNCPoint1[20795] = {X 427.7197, Y 45.9083, Z -2.1667, A 0.000, B 0.000, C 0.000 }
gfCNCPoint1[20796] = {X 427.6344, Y 45.0000, Z -2.1667, A 0.000, B 0.000, C 0.000 }
gfCNCPoint1[20797] = {X 427.6344, Y 44.2089, Z -2.1667, A 0.000, B 0.000, C 0.000 }
gfCNCPoint1[20798] = {X 427.7263, Y 43.2661, Z -2.1667, A 0.000, B 0.000, C 0.000 }
gfCNCPoint1[20799] = {X 427.9987, Y 42.3588, Z -2.1667, A 0.000, B 0.000, C 0.000 }
gfCNCPoint1[20800] = {X 428.4411, Y 41.5213, Z -2.1667, A 0.000, B 0.000, C 0.000 }
gfCNCPoint1[20801] = {X 429.0371, Y 40.7849, Z -2.1667, A 0.000, B 0.000, C 0.000 }
gfCNCPoint1[20802] = {X 429.7641, Y 40.1776, Z -2.1667, A 0.000, B 0.000, C 0.000 }
gfCNCPoint1[20803] = {X 430.5947, Y 39.7222, Z -2.1667, A 0.000, B 0.000, C 0.000 }
gfCNCPoint1[20804] = {X 434.2535, Y 32.5606, Z -2.1667, A 0.000, B 0.000, C 0.000 }
gfCNCPoint1[20805] = {X 432.9192, Y 31.5578, Z -2.1667, A 0.000, B 0.000, C 0.000 }
gfCNCPoint1[20806] = {X 431.7387, Y 30.3780, Z -2.1667, A 0.000, B 0.000, C 0.000 }
gfCNCPoint1[20807] = {X 430.7351, Y 29.0444, Z -2.1667, A 0.000, B 0.000, C 0.000 }
gfCNCPoint1[20808] = {X 429.9283, Y 27.5833, Z -2.1667, A 0.000, B 0.000, C 0.000 }
gfCNCPoint1[20809] = {X 429.3342, Y 26.0236, Z -2.1667, A 0.000, B 0.000, C 0.000 }
gfCNCPoint1[20810] = {X 428.9002, Y 24.1500, Z -2.1667, A 0.000, B 0.000, C 0.000 }
gfCNCPoint1[20811] = {X 428.6788, Y 22.2397, Z -2.1667, A 0.000, B 0.000, C 0.000 }
gfCNCPoint1[20812] = {X 428.6728, Y 20.3166, Z -2.1667, A 0.000, B 0.000, C 0.000 }
gfCNCPoint1[20813] = {X 428.8824, Y 18.4049, Z -2.1667, A 0.000, B 0.000, C 0.000 }
gfCNCPoint1[20814] = {X 429.3049, Y 16.5287, Z -2.1667, A 0.000, B 0.000, C 0.000 }
gfCNCPoint1[20815] = {X 429.8219, Y 15.0577, Z -2.1667, A 0.000, B 0.000, C 0.000 }
gfCNCPoint1[20816] = {X 430.5201, Y 13.6636, Z -2.1667, A 0.000, B 0.000, C 0.000 }
gfCNCPoint1[20817] = {X 431.3883, Y 12.3684, Z -2.1667, A 0.000, B 0.000, C 0.000 }
gfCNCPoint1[20818] = {X 432.4128, Y 11.1930, Z -2.1667, A 0.000, B 0.000, C 0.000 }
gfCNCPoint1[20819] = {X 433.6949, Y 10.0650, Z -2.1667, A 0.000, B 0.000, C 0.000 }
gfCNCPoint1[20820] = {X 435.1203, Y 9.1245, Z -2.1667, A 0.000, B 0.000, C 0.000 }
gfCNCPoint1[20821] = {X 436.6618, Y 8.3896, Z -2.1667, A 0.000, B 0.000, C 0.000 }
gfCNCPoint1[20822] = {X 438.2899, Y 7.8744, Z -2.1667, A 0.000, B 0.000, C 0.000 }
gfCNCPoint1[20823] = {X 439.9586, Y 7.5567, Z -2.1667, A 0.000, B 0.000, C 0.000 }
gfCNCPoint1[20824] = {X 441.6470, Y 7.3700, Z -2.1667, A 0.000, B 0.000, C 0.000 }
gfCNCPoint1[20825] = {X 443.3447, Y 7.3156, Z -2.1667, A 0.000, B 0.000, C 0.000 }
gfCNCPoint1[20826] = {X 444.0315, Y 7.3116, Z -2.1667, A 0.000, B 0.000, C 0.000 }
gfCNCPoint1[20827] = {X 459.4465, Y 7.3116, Z -2.1667, A 0.000, B 0.000, C 0.000 }
gfCNCPoint1[20828] = {X 460.4093, Y 7.4076, Z -2.1667, A 0.000, B 0.000, C 0.000 }
gfCNCPoint1[20829] = {X 461.3340, Y 7.6921, Z -2.1667, A 0.000, B 0.000, C 0.000 }
gfCNCPoint1[20830] = {X 462.1843, Y 8.1537, Z -2.1667, A 0.000, B 0.000, C 0.000 }
gfCNCPoint1[20831] = {X 462.9266, Y 8.7742, Z -2.1667, A 0.000, B 0.000, C 0.000 }
gfCNCPoint1[20832] = {X 463.5317, Y 9.5293, Z -2.1667, A 0.000, B 0.000, C 0.000 }
gfCNCPoint1[20833] = {X 463.9756, Y 10.3889, Z -2.1667, A 0.000, B 0.000, C 0.000 }
gfCNCPoint1[20834] = {X 464.2316, Y 11.2698, Z -2.1667, A 0.000, B 0.000, C 0.000 }
gfCNCPoint1[20835] = {X 464.3179, Y 12.1830, Z -2.1667, A 0.000, B 0.000, C 0.000 }
gfCNCPoint1[20836] = {X 464.3177, Y 13.0247, Z -2.1667, A 0.000, B 0.000, C 0.000 }
gfCNCPoint1[20837] = {X 464.2101, Y 13.9983, Z -2.1667, A 0.000, B 0.000, C 0.000 }
gfCNCPoint1[20838] = {X 463.9102, Y 14.9307, Z -2.1667, A 0.000, B 0.000, C 0.000 }
gfCNCPoint1[20839] = {X 463.4302, Y 15.7845, Z -2.1667, A 0.000, B 0.000, C 0.000 }
gfCNCPoint1[20840] = {X 462.7893, Y 16.5252, Z -2.1667, A 0.000, B 0.000, C 0.000 }
gfCNCPoint1[20841] = {X 462.7890, Y 16.7699, Z -2.1667, A 0.000, B 0.000, C 0.000 }
gfCNCPoint1[20842] = {X 462.7894, Y 25.8689, Z -2.1667, A 0.000, B 0.000, C 0.000 }
gfCNCPoint1[20843] = {X 467.5894, Y 25.8687, Z -2.1667, A 0.000, B 0.000, C 0.000 }
gfCNCPoint1[20844] = {X 467.5900, Y 38.9891, Z -2.1667, A 0.000, B 0.000, C 0.000 }
gfCNCPoint1[20845] = {X 467.6015, Y 39.0069, Z -2.1667, A 0.000, B 0.000, C 0.000 }
gfCNCPoint1[20846] = {X 468.3506, Y 37.9855, Z -2.1667, A 0.000, B 0.000, C 0.000 }
gfCNCPoint1[20847] = {X 469.2267, Y 37.0706, Z -2.1667, A 0.000, B 0.000, C 0.000 }
gfCNCPoint1[20848] = {X 470.2148, Y 36.2780, Z -2.1667, A 0.000, B 0.000, C 0.000 }
gfCNCPoint1[20849] = {X 471.5281, Y 33.7073, Z -2.1667, A 0.000, B 0.000, C 0.000 }
gfCNCPoint1[20850] = {X 470.4813, Y 32.4114, Z -2.1667, A 0.000, B 0.000, C 0.000 }
gfCNCPoint1[20851] = {X 469.5678, Y 31.0183, Z -2.1667, A 0.000, B 0.000, C 0.000 }
gfCNCPoint1[20852] = {X 468.7965, Y 29.5417, Z -2.1667, A 0.000, B 0.000, C 0.000 }
gfCNCPoint1[20853] = {X 468.1749, Y 27.9961, Z -2.1667, A 0.000, B 0.000, C 0.000 }
gfCNCPoint1[20854] = {X 467.7092, Y 26.3966, Z -2.1667, A 0.000, B 0.000, C 0.000 }
gfCNCPoint1[20855] = {X 467.6477, Y 26.1330, Z -2.1667, A 0.000, B 0.000, C 0.000 }
gfCNCPoint1[20856] = {X 467.5894, Y 25.8687, Z -2.1667, A 0.000, B 0.000, C 0.000 }
gfCNCPoint1[20857] = {X 465.1894, Y 25.8688, Z -2.1667, A 0.000, B 0.000, C 0.000 }
gfCNCPoint1[20858] = {X 465.1901, Y 39.7466, Z -2.1667, A 0.000, B 0.000, C 0.000 }
gfCNCPoint1[20859] = {X 465.3901, Y 40.0171, Z -2.1667, A 0.000, B 0.000, C 0.000 }
gfCNCPoint1[20860] = {X 465.5774, Y 40.2966, Z -2.1667, A 0.000, B 0.000, C 0.000 }
gfCNCPoint1[20861] = {X 466.0634, Y 41.1919, Z -2.1667, A 0.000, B 0.000, C 0.000 }
gfCNCPoint1[20862] = {X 466.4196, Y 42.1462, Z -2.1667, A 0.000, B 0.000, C 0.000 }
gfCNCPoint1[20863] = {X 466.6392, Y 43.1408, Z -2.1667, A 0.000, B 0.000, C 0.000 }
gfCNCPoint1[20864] = {X 466.7178, Y 44.1564, Z -2.1667, A 0.000, B 0.000, C 0.000 }
gfCNCPoint1[20865] = {X 466.7179, Y 45.0000, Z -2.1667, A 0.000, B 0.000, C 0.000 }
gfCNCPoint1[20866] = {X 466.7033, Y 45.4609, Z -2.1667, A 0.000, B 0.000, C 0.000 }
gfCNCPoint1[20867] = {X 466.6596, Y 45.9200, Z -2.1667, A 0.000, B 0.000, C 0.000 }
gfCNCPoint1[20868] = {X 468.5433, Y 45.9200, Z -2.1667, A 0.000, B 0.000, C 0.000 }
gfCNCPoint1[20869] = {X 468.4996, Y 45.4609, Z -2.1667, A 0.000, B 0.000, C 0.000 }
gfCNCPoint1[20870] = {X 468.4850, Y 45.0000, Z -2.1667, A 0.000, B 0.000, C 0.000 }
gfCNCPoint1[20871] = {X 468.4850, Y 44.2090, Z -2.1667, A 0.000, B 0.000, C 0.000 }
gfCNCPoint1[20872] = {X 468.5580, Y 43.1798, Z -2.1667, A 0.000, B 0.000, C 0.000 }
gfCNCPoint1[20873] = {X 468.7759, Y 42.1714, Z -2.1667, A 0.000, B 0.000, C 0.000 }
gfCNCPoint1[20874] = {X 469.1341, Y 41.2038, Z -2.1667, A 0.000, B 0.000, C 0.000 }
gfCNCPoint1[20875] = {X 469.6255, Y 40.2966, Z -2.1667, A 0.000, B 0.000, C 0.000 }
gfCNCPoint1[20876] = {X 470.3102, Y 39.3876, Z -2.1667, A 0.000, B 0.000, C 0.000 }
gfCNCPoint1[20877] = {X 471.1282, Y 38.5964, Z -2.1667, A 0.000, B 0.000, C 0.000 }
gfCNCPoint1[20878] = {X 472.0595, Y 37.9424, Z -2.1667, A 0.000, B 0.000, C 0.000 }
gfCNCPoint1[20879] = {X 474.4572, Y 33.2492, Z -2.1667, A 0.000, B 0.000, C 0.000 }
gfCNCPoint1[20880] = {X 473.2260, Y 32.0045, Z -2.1667, A 0.000, B 0.000, C 0.000 }
gfCNCPoint1[20881] = {X 472.1545, Y 30.6199, Z -2.1667, A 0.000, B 0.000, C 0.000 }
gfCNCPoint1[20882] = {X 471.2586, Y 29.1158, Z -2.1667, A 0.000, B 0.000, C 0.000 }
gfCNCPoint1[20883] = {X 470.5515, Y 27.5142, Z -2.1667, A 0.000, B 0.000, C 0.000 }
gfCNCPoint1[20884] = {X 470.0434, Y 25.8388, Z -2.1667, A 0.000, B 0.000, C 0.000 }
gfCNCPoint1[20885] = {X 469.9884, Y 25.6030, Z -2.1667, A 0.000, B 0.000, C 0.000 }
gfCNCPoint1[20886] = {X 469.9363, Y 25.3665, Z -2.1667, A 0.000, B 0.000, C 0.000 }
gfCNCPoint1[20887] = {X 469.6267, Y 23.4741, Z -2.1667, A 0.000, B 0.000, C 0.000 }
gfCNCPoint1[20888] = {X 469.5027, Y 21.5605, Z -2.1667, A 0.000, B 0.000, C 0.000 }
gfCNCPoint1[20889] = {X 469.5653, Y 19.6440, Z -2.1667, A 0.000, B 0.000, C 0.000 }
gfCNCPoint1[20890] = {X 469.8139, Y 17.7427, Z -2.1667, A 0.000, B 0.000, C 0.000 }
gfCNCPoint1[20891] = {X 470.2463, Y 15.8745, Z -2.1667, A 0.000, B 0.000, C 0.000 }
gfCNCPoint1[20892] = {X 470.6923, Y 14.5452, Z -2.1667, A 0.000, B 0.000, C 0.000 }
gfCNCPoint1[20893] = {X 471.2621, Y 13.2642, Z -2.1667, A 0.000, B 0.000, C 0.000 }
gfCNCPoint1[20894] = {X 469.1179, Y 12.1860, Z -2.1667, A 0.000, B 0.000, C 0.000 }
gfCNCPoint1[20895] = {X 469.1895, Y 12.0452, Z -2.1667, A 0.000, B 0.000, C 0.000 }
gfCNCPoint1[20896] = {X 469.2624, Y 11.9051, Z -2.1667, A 0.000, B 0.000, C 0.000 }
gfCNCPoint1[20897] = {X 469.1139, Y 11.9051, Z -2.1667, A 0.000, B 0.000, C 0.000 }
gfCNCPoint1[20898] = {X 469.1170, Y 12.0455, Z -2.1667, A 0.000, B 0.000, C 0.000 }
gfCNCPoint1[20899] = {X 469.1179, Y 12.1860, Z -2.1667, A 0.000, B 0.000, C 0.000 }
gfCNCPoint1[20900] = {X 471.2621, Y 13.2642, Z -2.1667, A 0.000, B 0.000, C 0.000 }
gfCNCPoint1[20901] = {X 471.3237, Y 13.1430, Z -2.1667, A 0.000, B 0.000, C 0.000 }
gfCNCPoint1[20902] = {X 471.3865, Y 13.0225, Z -2.1667, A 0.000, B 0.000, C 0.000 }
gfCNCPoint1[20903] = {X 472.1280, Y 11.7671, Z -2.1667, A 0.000, B 0.000, C 0.000 }
gfCNCPoint1[20904] = {X 472.9895, Y 10.5909, Z -2.1667, A 0.000, B 0.000, C 0.000 }
gfCNCPoint1[20905] = {X 473.9626, Y 9.5051, Z -2.1667, A 0.000, B 0.000, C 0.000 }
gfCNCPoint1[20906] = {X 466.2069, Y 9.5051, Z -2.1667, A 0.000, B 0.000, C 0.000 }
gfCNCPoint1[20907] = {X 466.5687, Y 10.7174, Z -2.1667, A 0.000, B 0.000, C 0.000 }
gfCNCPoint1[20908] = {X 466.7149, Y 11.9740, Z -2.1667, A 0.000, B 0.000, C 0.000 }
gfCNCPoint1[20909] = {X 466.7172, Y 12.0785, Z -2.1667, A 0.000, B 0.000, C 0.000 }
gfCNCPoint1[20910] = {X 466.7179, Y 12.1830, Z -2.1667, A 0.000, B 0.000, C 0.000 }
gfCNCPoint1[20911] = {X 466.7176, Y 13.0477, Z -2.1667, A 0.000, B 0.000, C 0.000 }
gfCNCPoint1[20912] = {X 466.6103, Y 14.2253, Z -2.1667, A 0.000, B 0.000, C 0.000 }
gfCNCPoint1[20913] = {X 466.3137, Y 15.3700, Z -2.1667, A 0.000, B 0.000, C 0.000 }
gfCNCPoint1[20914] = {X 465.8358, Y 16.4516, Z -2.1667, A 0.000, B 0.000, C 0.000 }
gfCNCPoint1[20915] = {X 465.1890, Y 17.4416, Z -2.1667, A 0.000, B 0.000, C 0.000 }
gfCNCPoint1[20916] = {X 465.1894, Y 25.8688, Z -2.1667, A 0.000, B 0.000, C 0.000 }
gfCNCPoint1[20917] = {X 462.7894, Y 25.8689, Z -2.1667, A 0.000, B 0.000, C 0.000 }
gfCNCPoint1[20918] = {X 462.7901, Y 40.6624, Z -2.1667, A 0.000, B 0.000, C 0.000 }
gfCNCPoint1[20919] = {X 463.4314, Y 41.4040, Z -2.1667, A 0.000, B 0.000, C 0.000 }
gfCNCPoint1[20920] = {X 463.9114, Y 42.2588, Z -2.1667, A 0.000, B 0.000, C 0.000 }
gfCNCPoint1[20921] = {X 464.2109, Y 43.1924, Z -2.1667, A 0.000, B 0.000, C 0.000 }
gfCNCPoint1[20922] = {X 464.3178, Y 44.1670, Z -2.1667, A 0.000, B 0.000, C 0.000 }
gfCNCPoint1[20923] = {X 464.3179, Y 45.0000, Z -2.1667, A 0.000, B 0.000, C 0.000 }
gfCNCPoint1[20924] = {X 464.3081, Y 45.3090, Z -2.1667, A 0.000, B 0.000, C 0.000 }
gfCNCPoint1[20925] = {X 464.2788, Y 45.6167, Z -2.1667, A 0.000, B 0.000, C 0.000 }
gfCNCPoint1[20926] = {X 464.0485, Y 46.5992, Z -2.1667, A 0.000, B 0.000, C 0.000 }
gfCNCPoint1[20927] = {X 463.6209, Y 47.5134, Z -2.1667, A 0.000, B 0.000, C 0.000 }
gfCNCPoint1[20928] = {X 463.0145, Y 48.3200, Z -2.1667, A 0.000, B 0.000, C 0.000 }
gfCNCPoint1[20929] = {X 462.6627, Y 47.9934, Z -2.1667, A 0.000, B 0.000, C 0.000 }
gfCNCPoint1[20930] = {X 461.9835, Y 48.5889, Z -2.1667, A 0.000, B 0.000, C 0.000 }
gfCNCPoint1[20931] = {X 461.1970, Y 49.0331, Z -2.1667, A 0.000, B 0.000, C 0.000 }
gfCNCPoint1[20932] = {X 460.3364, Y 49.3073, Z -2.1667, A 0.000, B 0.000, C 0.000 }
gfCNCPoint1[20933] = {X 459.4379, Y 49.4000, Z -2.1667, A 0.000, B 0.000, C 0.000 }
gfCNCPoint1[20934] = {X 452.9945, Y 49.4000, Z -2.1667, A 0.000, B 0.000, C 0.000 }
gfCNCPoint1[20935] = {X 452.0154, Y 49.2897, Z -2.1667, A 0.000, B 0.000, C 0.000 }
gfCNCPoint1[20936] = {X 451.0854, Y 48.9643, Z -2.1667, A 0.000, B 0.000, C 0.000 }
gfCNCPoint1[20937] = {X 450.2511, Y 48.4400, Z -2.1667, A 0.000, B 0.000, C 0.000 }
gfCNCPoint1[20938] = {X 449.5544, Y 47.7433, Z -2.1667, A 0.000, B 0.000, C 0.000 }
gfCNCPoint1[20939] = {X 449.0302, Y 46.9091, Z -2.1667, A 0.000, B 0.000, C 0.000 }
gfCNCPoint1[20940] = {X 448.7048, Y 45.9791, Z -2.1667, A 0.000, B 0.000, C 0.000 }
gfCNCPoint1[20941] = {X 448.5945, Y 45.0000, Z -2.1667, A 0.000, B 0.000, C 0.000 }
gfCNCPoint1[20942] = {X 448.5949, Y 44.1483, Z -2.1667, A 0.000, B 0.000, C 0.000 }
gfCNCPoint1[20943] = {X 448.7053, Y 43.2275, Z -2.1667, A 0.000, B 0.000, C 0.000 }
gfCNCPoint1[20944] = {X 449.0063, Y 42.3503, Z -2.1667, A 0.000, B 0.000, C 0.000 }
gfCNCPoint1[20945] = {X 449.4844, Y 41.5556, Z -2.1667, A 0.000, B 0.000, C 0.000 }
gfCNCPoint1[20946] = {X 450.1184, Y 40.8789, Z -2.1667, A 0.000, B 0.000, C 0.000 }
gfCNCPoint1[20947] = {X 450.1184, Y 34.5538, Z -2.1667, A 0.000, B 0.000, C 0.000 }
gfCNCPoint1[20948] = {X 447.5225, Y 34.5538, Z -2.1667, A 0.000, B 0.000, C 0.000 }
gfCNCPoint1[20949] = {X 443.2761, Y 42.8215, Z -2.1667, A 0.000, B 0.000, C 0.000 }
gfCNCPoint1[20950] = {X 443.4440, Y 43.5062, Z -2.1667, A 0.000, B 0.000, C 0.000 }
gfCNCPoint1[20951] = {X 443.5005, Y 44.2089, Z -2.1667, A 0.000, B 0.000, C 0.000 }
gfCNCPoint1[20952] = {X 443.5005, Y 45.0000, Z -2.1667, A 0.000, B 0.000, C 0.000 }
gfCNCPoint1[20953] = {X 443.3902, Y 45.9791, Z -2.1667, A 0.000, B 0.000, C 0.000 }
gfCNCPoint1[20954] = {X 443.0647, Y 46.9091, Z -2.1667, A 0.000, B 0.000, C 0.000 }
gfCNCPoint1[20955] = {X 442.5405, Y 47.7434, Z -2.1667, A 0.000, B 0.000, C 0.000 }
gfCNCPoint1[20956] = {X 441.8438, Y 48.4401, Z -2.1667, A 0.000, B 0.000, C 0.000 }
gfCNCPoint1[20957] = {X 441.0096, Y 48.9643, Z -2.1667, A 0.000, B 0.000, C 0.000 }
gfCNCPoint1[20958] = {X 440.0796, Y 49.2897, Z -2.1667, A 0.000, B 0.000, C 0.000 }
gfCNCPoint1[20959] = {X 439.1005, Y 49.4000, Z -2.1667, A 0.000, B 0.000, C 0.000 }
gfCNCPoint1[20960] = {X 432.5144, Y 49.4000, Z -2.1667, A 0.000, B 0.000, C 0.000 }
gfCNCPoint1[20961] = {X 431.5353, Y 49.2897, Z -2.1667, A 0.000, B 0.000, C 0.000 }
gfCNCPoint1[20962] = {X 430.6053, Y 48.9643, Z -2.1667, A 0.000, B 0.000, C 0.000 }
gfCNCPoint1[20963] = {X 429.7711, Y 48.4401, Z -2.1667, A 0.000, B 0.000, C 0.000 }
gfCNCPoint1[20964] = {X 429.0743, Y 47.7434, Z -2.1667, A 0.000, B 0.000, C 0.000 }
gfCNCPoint1[20965] = {X 428.5501, Y 46.9091, Z -2.1667, A 0.000, B 0.000, C 0.000 }
gfCNCPoint1[20966] = {X 428.2247, Y 45.9791, Z -2.1667, A 0.000, B 0.000, C 0.000 }
gfCNCPoint1[20967] = {X 428.1144, Y 45.0000, Z -2.1667, A 0.000, B 0.000, C 0.000 }
gfCNCPoint1[20968] = {X 428.1148, Y 44.1483, Z -2.1667, A 0.000, B 0.000, C 0.000 }
gfCNCPoint1[20969] = {X 428.2132, Y 43.2816, Z -2.1667, A 0.000, B 0.000, C 0.000 }
gfCNCPoint1[20970] = {X 428.4806, Y 42.4514, Z -2.1667, A 0.000, B 0.000, C 0.000 }
gfCNCPoint1[20971] = {X 428.9065, Y 41.6903, Z -2.1667, A 0.000, B 0.000, C 0.000 }
gfCNCPoint1[20972] = {X 429.4741, Y 41.0281, Z -2.1667, A 0.000, B 0.000, C 0.000 }
gfCNCPoint1[20973] = {X 430.1613, Y 40.4909, Z -2.1667, A 0.000, B 0.000, C 0.000 }
gfCNCPoint1[20974] = {X 430.9408, Y 40.0998, Z -2.1667, A 0.000, B 0.000, C 0.000 }
gfCNCPoint1[20975] = {X 434.8819, Y 32.3856, Z -2.1667, A 0.000, B 0.000, C 0.000 }
gfCNCPoint1[20976] = {X 433.7185, Y 31.5931, Z -2.1667, A 0.000, B 0.000, C 0.000 }
gfCNCPoint1[20977] = {X 432.6616, Y 30.6632, Z -2.1667, A 0.000, B 0.000, C 0.000 }
gfCNCPoint1[20978] = {X 431.7274, Y 29.6102, Z -2.1667, A 0.000, B 0.000, C 0.000 }
gfCNCPoint1[20979] = {X 430.9301, Y 28.4501, Z -2.1667, A 0.000, B 0.000, C 0.000 }
gfCNCPoint1[20980] = {X 430.2818, Y 27.2006, Z -2.1667, A 0.000, B 0.000, C 0.000 }
gfCNCPoint1[20981] = {X 429.7925, Y 25.8807, Z -2.1667, A 0.000, B 0.000, C 0.000 }
gfCNCPoint1[20982] = {X 429.3719, Y 24.0610, Z -2.1667, A 0.000, B 0.000, C 0.000 }
gfCNCPoint1[20983] = {X 429.1576, Y 22.2057, Z -2.1667, A 0.000, B 0.000, C 0.000 }
gfCNCPoint1[20984] = {X 429.1523, Y 20.3381, Z -2.1667, A 0.000, B 0.000, C 0.000 }
gfCNCPoint1[20985] = {X 429.3562, Y 18.4816, Z -2.1667, A 0.000, B 0.000, C 0.000 }
gfCNCPoint1[20986] = {X 429.7667, Y 16.6596, Z -2.1667, A 0.000, B 0.000, C 0.000 }
gfCNCPoint1[20987] = {X 430.2919, Y 15.1794, Z -2.1667, A 0.000, B 0.000, C 0.000 }
gfCNCPoint1[20988] = {X 431.0078, Y 13.7815, Z -2.1667, A 0.000, B 0.000, C 0.000 }
gfCNCPoint1[20989] = {X 431.9021, Y 12.4903, Z -2.1667, A 0.000, B 0.000, C 0.000 }
gfCNCPoint1[20990] = {X 432.9589, Y 11.3285, Z -2.1667, A 0.000, B 0.000, C 0.000 }
gfCNCPoint1[20991] = {X 434.1599, Y 10.3163, Z -2.1667, A 0.000, B 0.000, C 0.000 }
gfCNCPoint1[20992] = {X 435.4839, Y 9.4715, Z -2.1667, A 0.000, B 0.000, C 0.000 }
gfCNCPoint1[20993] = {X 436.9079, Y 8.8088, Z -2.1667, A 0.000, B 0.000, C 0.000 }
gfCNCPoint1[20994] = {X 438.4069, Y 8.3400, Z -2.1667, A 0.000, B 0.000, C 0.000 }
gfCNCPoint1[20995] = {X 440.0369, Y 8.0303, Z -2.1667, A 0.000, B 0.000, C 0.000 }
gfCNCPoint1[20996] = {X 441.6861, Y 7.8484, Z -2.1667, A 0.000, B 0.000, C 0.000 }
gfCNCPoint1[20997] = {X 443.3444, Y 7.7956, Z -2.1667, A 0.000, B 0.000, C 0.000 }
gfCNCPoint1[20998] = {X 444.0367, Y 7.7916, Z -2.1667, A 0.000, B 0.000, C 0.000 }
gfCNCPoint1[20999] = {X 459.4465, Y 7.7916, Z -2.1667, A 0.000, B 0.000, C 0.000 }
gfCNCPoint1[21000] = {X 460.4237, Y 7.9017, Z -2.1667, A 0.000, B 0.000, C 0.000 }
gfCNCPoint1[21001] = {X 461.3519, Y 8.2265, Z -2.1667, A 0.000, B 0.000, C 0.000 }
gfCNCPoint1[21002] = {X 462.1845, Y 8.7496, Z -2.1667, A 0.000, B 0.000, C 0.000 }
gfCNCPoint1[21003] = {X 462.8799, Y 9.4450, Z -2.1667, A 0.000, B 0.000, C 0.000 }
gfCNCPoint1[21004] = {X 463.4031, Y 10.2776, Z -2.1667, A 0.000, B 0.000, C 0.000 }
gfCNCPoint1[21005] = {X 463.7278, Y 11.2058, Z -2.1667, A 0.000, B 0.000, C 0.000 }
gfCNCPoint1[21006] = {X 463.8379, Y 12.1830, Z -2.1667, A 0.000, B 0.000, C 0.000 }
gfCNCPoint1[21007] = {X 463.8377, Y 13.0201, Z -2.1667, A 0.000, B 0.000, C 0.000 }
gfCNCPoint1[21008] = {X 463.7299, Y 13.9473, Z -2.1667, A 0.000, B 0.000, C 0.000 }
gfCNCPoint1[21009] = {X 463.4288, Y 14.8308, Z -2.1667, A 0.000, B 0.000, C 0.000 }
gfCNCPoint1[21010] = {X 462.9482, Y 15.6310, Z -2.1667, A 0.000, B 0.000, C 0.000 }
gfCNCPoint1[21011] = {X 462.3096, Y 16.3118, Z -2.1667, A 0.000, B 0.000, C 0.000 }
gfCNCPoint1[21012] = {X 462.3090, Y 16.7692, Z -2.1667, A 0.000, B 0.000, C 0.000 }
gfCNCPoint1[21013] = {X 462.3101, Y 40.8756, Z -2.1667, A 0.000, B 0.000, C 0.000 }
gfCNCPoint1[21014] = {X 462.9549, Y 41.5647, Z -2.1667, A 0.000, B 0.000, C 0.000 }
gfCNCPoint1[21015] = {X 463.4378, Y 42.3755, Z -2.1667, A 0.000, B 0.000, C 0.000 }
gfCNCPoint1[21016] = {X 463.7368, Y 43.2706, Z -2.1667, A 0.000, B 0.000, C 0.000 }
gfCNCPoint1[21017] = {X 463.8379, Y 44.2089, Z -2.1667, A 0.000, B 0.000, C 0.000 }
gfCNCPoint1[21018] = {X 463.8379, Y 45.0000, Z -2.1667, A 0.000, B 0.000, C 0.000 }
gfCNCPoint1[21019] = {X 463.7612, Y 45.8182, Z -2.1667, A 0.000, B 0.000, C 0.000 }
gfCNCPoint1[21020] = {X 463.5336, Y 46.6079, Z -2.1667, A 0.000, B 0.000, C 0.000 }
gfCNCPoint1[21021] = {X 463.1632, Y 47.3415, Z -2.1667, A 0.000, B 0.000, C 0.000 }
gfCNCPoint1[21022] = {X 462.6627, Y 47.9934, Z -2.1667, A 0.000, B 0.000, C 0.000 }
gfCNCPoint1[21023] = {X 463.0145, Y 48.3200, Z -2.1667, A 0.000, B 0.000, C 0.000 }
gfCNCPoint1[21024] = {X 472.1884, Y 48.3200, Z -2.1667, A 0.000, B 0.000, C 0.000 }
gfCNCPoint1[21025] = {X 471.5820, Y 47.5134, Z -2.1667, A 0.000, B 0.000, C 0.000 }
gfCNCPoint1[21026] = {X 471.1544, Y 46.5992, Z -2.1667, A 0.000, B 0.000, C 0.000 }
gfCNCPoint1[21027] = {X 470.9241, Y 45.6167, Z -2.1667, A 0.000, B 0.000, C 0.000 }
gfCNCPoint1[21028] = {X 470.8947, Y 45.3090, Z -2.1667, A 0.000, B 0.000, C 0.000 }
gfCNCPoint1[21029] = {X 470.8850, Y 45.0000, Z -2.1667, A 0.000, B 0.000, C 0.000 }
gfCNCPoint1[21030] = {X 470.8850, Y 44.2089, Z -2.1667, A 0.000, B 0.000, C 0.000 }
gfCNCPoint1[21031] = {X 470.9769, Y 43.2661, Z -2.1667, A 0.000, B 0.000, C 0.000 }
gfCNCPoint1[21032] = {X 471.2492, Y 42.3588, Z -2.1667, A 0.000, B 0.000, C 0.000 }
gfCNCPoint1[21033] = {X 471.6917, Y 41.5212, Z -2.1667, A 0.000, B 0.000, C 0.000 }
gfCNCPoint1[21034] = {X 472.2877, Y 40.7849, Z -2.1667, A 0.000, B 0.000, C 0.000 }
gfCNCPoint1[21035] = {X 473.0146, Y 40.1776, Z -2.1667, A 0.000, B 0.000, C 0.000 }
gfCNCPoint1[21036] = {X 473.8453, Y 39.7222, Z -2.1667, A 0.000, B 0.000, C 0.000 }
gfCNCPoint1[21037] = {X 477.5004, Y 32.5678, Z -2.1667, A 0.000, B 0.000, C 0.000 }
gfCNCPoint1[21038] = {X 476.2833, Y 31.6577, Z -2.1667, A 0.000, B 0.000, C 0.000 }
gfCNCPoint1[21039] = {X 475.1907, Y 30.6015, Z -2.1667, A 0.000, B 0.000, C 0.000 }
gfCNCPoint1[21040] = {X 474.2399, Y 29.4159, Z -2.1667, A 0.000, B 0.000, C 0.000 }
gfCNCPoint1[21041] = {X 473.4461, Y 28.1200, Z -2.1667, A 0.000, B 0.000, C 0.000 }
gfCNCPoint1[21042] = {X 472.8221, Y 26.7343, Z -2.1667, A 0.000, B 0.000, C 0.000 }
gfCNCPoint1[21043] = {X 472.3777, Y 25.2810, Z -2.1667, A 0.000, B 0.000, C 0.000 }
gfCNCPoint1[21044] = {X 472.0534, Y 23.5417, Z -2.1667, A 0.000, B 0.000, C 0.000 }
gfCNCPoint1[21045] = {X 471.9084, Y 21.7784, Z -2.1667, A 0.000, B 0.000, C 0.000 }
gfCNCPoint1[21046] = {X 471.9443, Y 20.0095, Z -2.1667, A 0.000, B 0.000, C 0.000 }
gfCNCPoint1[21047] = {X 472.1607, Y 18.2535, Z -2.1667, A 0.000, B 0.000, C 0.000 }
gfCNCPoint1[21048] = {X 472.5554, Y 16.5288, Z -2.1667, A 0.000, B 0.000, C 0.000 }
gfCNCPoint1[21049] = {X 473.0746, Y 15.0579, Z -2.1667, A 0.000, B 0.000, C 0.000 }
gfCNCPoint1[21050] = {X 473.7744, Y 13.6638, Z -2.1667, A 0.000, B 0.000, C 0.000 }
gfCNCPoint1[21051] = {X 474.6437, Y 12.3687, Z -2.1667, A 0.000, B 0.000, C 0.000 }
gfCNCPoint1[21052] = {X 475.6688, Y 11.1929, Z -2.1667, A 0.000, B 0.000, C 0.000 }
gfCNCPoint1[21053] = {X 476.7459, Y 10.2244, Z -2.1667, A 0.000, B 0.000, C 0.000 }
gfCNCPoint1[21054] = {X 477.9286, Y 9.3882, Z -2.1667, A 0.000, B 0.000, C 0.000 }
gfCNCPoint1[21055] = {X 479.2007, Y 8.6956, Z -2.1667, A 0.000, B 0.000, C 0.000 }
gfCNCPoint1[21056] = {X 480.5450, Y 8.1561, Z -2.1667, A 0.000, B 0.000, C 0.000 }
gfCNCPoint1[21057] = {X 481.9430, Y 7.7771, Z -2.1667, A 0.000, B 0.000, C 0.000 }
gfCNCPoint1[21058] = {X 484.0944, Y 7.4422, Z -2.1667, A 0.000, B 0.000, C 0.000 }
gfCNCPoint1[21059] = {X 486.2685, Y 7.3238, Z -2.1667, A 0.000, B 0.000, C 0.000 }
gfCNCPoint1[21060] = {X 486.9707, Y 7.3116, Z -2.1667, A 0.000, B 0.000, C 0.000 }
gfCNCPoint1[21061] = {X 502.2122, Y 7.3116, Z -2.1667, A 0.000, B 0.000, C 0.000 }
gfCNCPoint1[21062] = {X 502.7417, Y 7.3157, Z -2.1667, A 0.000, B 0.000, C 0.000 }
gfCNCPoint1[21063] = {X 503.6962, Y 7.4179, Z -2.1667, A 0.000, B 0.000, C 0.000 }
gfCNCPoint1[21064] = {X 504.6120, Y 7.7055, Z -2.1667, A 0.000, B 0.000, C 0.000 }
gfCNCPoint1[21065] = {X 505.4535, Y 8.1673, Z -2.1667, A 0.000, B 0.000, C 0.000 }
gfCNCPoint1[21066] = {X 506.1880, Y 8.7854, Z -2.1667, A 0.000, B 0.000, C 0.000 }
gfCNCPoint1[21067] = {X 506.7868, Y 9.5357, Z -2.1667, A 0.000, B 0.000, C 0.000 }
gfCNCPoint1[21068] = {X 507.2266, Y 10.3889, Z -2.1667, A 0.000, B 0.000, C 0.000 }
gfCNCPoint1[21069] = {X 507.4823, Y 11.2685, Z -2.1667, A 0.000, B 0.000, C 0.000 }
gfCNCPoint1[21070] = {X 507.5685, Y 12.1804, Z -2.1667, A 0.000, B 0.000, C 0.000 }
gfCNCPoint1[21071] = {X 507.5683, Y 13.0237, Z -2.1667, A 0.000, B 0.000, C 0.000 }
gfCNCPoint1[21072] = {X 507.4608, Y 13.9974, Z -2.1667, A 0.000, B 0.000, C 0.000 }
gfCNCPoint1[21073] = {X 507.1611, Y 14.9300, Z -2.1667, A 0.000, B 0.000, C 0.000 }
gfCNCPoint1[21074] = {X 506.6811, Y 15.7839, Z -2.1667, A 0.000, B 0.000, C 0.000 }
gfCNCPoint1[21075] = {X 506.0403, Y 16.5248, Z -2.1667, A 0.000, B 0.000, C 0.000 }
gfCNCPoint1[21076] = {X 506.0402, Y 40.6619, Z -2.1667, A 0.000, B 0.000, C 0.000 }
gfCNCPoint1[21077] = {X 506.6816, Y 41.4035, Z -2.1667, A 0.000, B 0.000, C 0.000 }
gfCNCPoint1[21078] = {X 507.1617, Y 42.2583, Z -2.1667, A 0.000, B 0.000, C 0.000 }
gfCNCPoint1[21079] = {X 507.4614, Y 43.1919, Z -2.1667, A 0.000, B 0.000, C 0.000 }
gfCNCPoint1[21080] = {X 507.5683, Y 44.1665, Z -2.1667, A 0.000, B 0.000, C 0.000 }
gfCNCPoint1[21081] = {X 507.5685, Y 45.0000, Z -2.1667, A 0.000, B 0.000, C 0.000 }
gfCNCPoint1[21082] = {X 507.4747, Y 45.9520, Z -2.1667, A 0.000, B 0.000, C 0.000 }
gfCNCPoint1[21083] = {X 507.1970, Y 46.8675, Z -2.1667, A 0.000, B 0.000, C 0.000 }
gfCNCPoint1[21084] = {X 506.7461, Y 47.7112, Z -2.1667, A 0.000, B 0.000, C 0.000 }
gfCNCPoint1[21085] = {X 506.1392, Y 48.4507, Z -2.1667, A 0.000, B 0.000, C 0.000 }
gfCNCPoint1[21086] = {X 505.3997, Y 49.0576, Z -2.1667, A 0.000, B 0.000, C 0.000 }
gfCNCPoint1[21087] = {X 504.5560, Y 49.5085, Z -2.1667, A 0.000, B 0.000, C 0.000 }
gfCNCPoint1[21088] = {X 503.6405, Y 49.7862, Z -2.1667, A 0.000, B 0.000, C 0.000 }
gfCNCPoint1[21089] = {X 502.6885, Y 49.8800, Z -2.1667, A 0.000, B 0.000, C 0.000 }
gfCNCPoint1[21090] = {X 496.2450, Y 49.8800, Z -2.1667, A 0.000, B 0.000, C 0.000 }
gfCNCPoint1[21091] = {X 495.2220, Y 49.7716, Z -2.1667, A 0.000, B 0.000, C 0.000 }
gfCNCPoint1[21092] = {X 494.2445, Y 49.4511, Z -2.1667, A 0.000, B 0.000, C 0.000 }
gfCNCPoint1[21093] = {X 493.3559, Y 48.9328, Z -2.1667, A 0.000, B 0.000, C 0.000 }
gfCNCPoint1[21094] = {X 492.5956, Y 48.2398, Z -2.1667, A 0.000, B 0.000, C 0.000 }
gfCNCPoint1[21095] = {X 491.9976, Y 47.4028, Z -2.1667, A 0.000, B 0.000, C 0.000 }
gfCNCPoint1[21096] = {X 491.5882, Y 46.4590, Z -2.1667, A 0.000, B 0.000, C 0.000 }
gfCNCPoint1[21097] = {X 491.4241, Y 45.7570, Z -2.1667, A 0.000, B 0.000, C 0.000 }
gfCNCPoint1[21098] = {X 491.3652, Y 45.0385, Z -2.1667, A 0.000, B 0.000, C 0.000 }
gfCNCPoint1[21099] = {X 491.3655, Y 44.1416, Z -2.1667, A 0.000, B 0.000, C 0.000 }
gfCNCPoint1[21100] = {X 491.4758, Y 43.1751, Z -2.1667, A 0.000, B 0.000, C 0.000 }
gfCNCPoint1[21101] = {X 491.7756, Y 42.2497, Z -2.1667, A 0.000, B 0.000, C 0.000 }
gfCNCPoint1[21102] = {X 492.2530, Y 41.4020, Z -2.1667, A 0.000, B 0.000, C 0.000 }
gfCNCPoint1[21103] = {X 492.8890, Y 40.6660, Z -2.1667, A 0.000, B 0.000, C 0.000 }
gfCNCPoint1[21104] = {X 492.8890, Y 35.0338, Z -2.1667, A 0.000, B 0.000, C 0.000 }
gfCNCPoint1[21105] = {X 491.0654, Y 35.0338, Z -2.1667, A 0.000, B 0.000, C 0.000 }
gfCNCPoint1[21106] = {X 487.0429, Y 42.8669, Z -2.1667, A 0.000, B 0.000, C 0.000 }
gfCNCPoint1[21107] = {X 487.1807, Y 43.5095, Z -2.1667, A 0.000, B 0.000, C 0.000 }
gfCNCPoint1[21108] = {X 487.2308, Y 44.1648, Z -2.1667, A 0.000, B 0.000, C 0.000 }
gfCNCPoint1[21109] = {X 487.2310, Y 45.0000, Z -2.1667, A 0.000, B 0.000, C 0.000 }
gfCNCPoint1[21110] = {X 487.1749, Y 45.7380, Z -2.1667, A 0.000, B 0.000, C 0.000 }
gfCNCPoint1[21111] = {X 487.0078, Y 46.4590, Z -2.1667, A 0.000, B 0.000, C 0.000 }
gfCNCPoint1[21112] = {X 486.5939, Y 47.4110, Z -2.1667, A 0.000, B 0.000, C 0.000 }
gfCNCPoint1[21113] = {X 485.9879, Y 48.2538, Z -2.1667, A 0.000, B 0.000, C 0.000 }
gfCNCPoint1[21114] = {X 485.2175, Y 48.9494, Z -2.1667, A 0.000, B 0.000, C 0.000 }
gfCNCPoint1[21115] = {X 484.3173, Y 49.4663, Z -2.1667, A 0.000, B 0.000, C 0.000 }
gfCNCPoint1[21116] = {X 483.3557, Y 49.7755, Z -2.1667, A 0.000, B 0.000, C 0.000 }
gfCNCPoint1[21117] = {X 482.3510, Y 49.8800, Z -2.1667, A 0.000, B 0.000, C 0.000 }
gfCNCPoint1[21118] = {X 480.2695, Y 49.8800, Z -2.1667, A 0.000, B 0.000, C 0.000 }
gfCNCPoint1[21119] = {X 480.2695, Y 49.4000, Z -2.1667, A 0.000, B 0.000, C 0.000 }
gfCNCPoint1[21120] = {X 475.7650, Y 49.4000, Z -2.1667, A 0.000, B 0.000, C 0.000 }
gfCNCPoint1[21121] = {X 474.7859, Y 49.2897, Z -2.1667, A 0.000, B 0.000, C 0.000 }
gfCNCPoint1[21122] = {X 473.8559, Y 48.9643, Z -2.1667, A 0.000, B 0.000, C 0.000 }
gfCNCPoint1[21123] = {X 473.0216, Y 48.4401, Z -2.1667, A 0.000, B 0.000, C 0.000 }
gfCNCPoint1[21124] = {X 472.3249, Y 47.7434, Z -2.1667, A 0.000, B 0.000, C 0.000 }
gfCNCPoint1[21125] = {X 471.8007, Y 46.9091, Z -2.1667, A 0.000, B 0.000, C 0.000 }
gfCNCPoint1[21126] = {X 471.4753, Y 45.9791, Z -2.1667, A 0.000, B 0.000, C 0.000 }
gfCNCPoint1[21127] = {X 471.3650, Y 45.0000, Z -2.1667, A 0.000, B 0.000, C 0.000 }
gfCNCPoint1[21128] = {X 471.3654, Y 44.1483, Z -2.1667, A 0.000, B 0.000, C 0.000 }
gfCNCPoint1[21129] = {X 471.4638, Y 43.2816, Z -2.1667, A 0.000, B 0.000, C 0.000 }
gfCNCPoint1[21130] = {X 471.7311, Y 42.4514, Z -2.1667, A 0.000, B 0.000, C 0.000 }
gfCNCPoint1[21131] = {X 472.1570, Y 41.6903, Z -2.1667, A 0.000, B 0.000, C 0.000 }
gfCNCPoint1[21132] = {X 472.7247, Y 41.0281, Z -2.1667, A 0.000, B 0.000, C 0.000 }
gfCNCPoint1[21133] = {X 473.4118, Y 40.4909, Z -2.1667, A 0.000, B 0.000, C 0.000 }
gfCNCPoint1[21134] = {X 474.1914, Y 40.0998, Z -2.1667, A 0.000, B 0.000, C 0.000 }
gfCNCPoint1[21135] = {X 478.1278, Y 32.3948, Z -2.1667, A 0.000, B 0.000, C 0.000 }
gfCNCPoint1[21136] = {X 476.8712, Y 31.5205, Z -2.1667, A 0.000, B 0.000, C 0.000 }
gfCNCPoint1[21137] = {X 475.7413, Y 30.4878, Z -2.1667, A 0.000, B 0.000, C 0.000 }
gfCNCPoint1[21138] = {X 474.7579, Y 29.3147, Z -2.1667, A 0.000, B 0.000, C 0.000 }
gfCNCPoint1[21139] = {X 473.9382, Y 28.0219, Z -2.1667, A 0.000, B 0.000, C 0.000 }
gfCNCPoint1[21140] = {X 473.2967, Y 26.6320, Z -2.1667, A 0.000, B 0.000, C 0.000 }
gfCNCPoint1[21141] = {X 472.8446, Y 25.1695, Z -2.1667, A 0.000, B 0.000, C 0.000 }
gfCNCPoint1[21142] = {X 472.5292, Y 23.4784, Z -2.1667, A 0.000, B 0.000, C 0.000 }
gfCNCPoint1[21143] = {X 472.3882, Y 21.7639, Z -2.1667, A 0.000, B 0.000, C 0.000 }
gfCNCPoint1[21144] = {X 472.4230, Y 20.0440, Z -2.1667, A 0.000, B 0.000, C 0.000 }
gfCNCPoint1[21145] = {X 472.6335, Y 18.3366, Z -2.1667, A 0.000, B 0.000, C 0.000 }
gfCNCPoint1[21146] = {X 473.0172, Y 16.6597, Z -2.1667, A 0.000, B 0.000, C 0.000 }
gfCNCPoint1[21147] = {X 473.5641, Y 15.1350, Z -2.1667, A 0.000, B 0.000, C 0.000 }
gfCNCPoint1[21148] = {X 474.3127, Y 13.6986, Z -2.1667, A 0.000, B 0.000, C 0.000 }
gfCNCPoint1[21149] = {X 475.2492, Y 12.3769, Z -2.1667, A 0.000, B 0.000, C 0.000 }
gfCNCPoint1[21150] = {X 476.3562, Y 11.1944, Z -2.1667, A 0.000, B 0.000, C 0.000 }
gfCNCPoint1[21151] = {X 477.6134, Y 10.1730, Z -2.1667, A 0.000, B 0.000, C 0.000 }
gfCNCPoint1[21152] = {X 478.9974, Y 9.3315, Z -2.1667, A 0.000, B 0.000, C 0.000 }
gfCNCPoint1[21153] = {X 480.4828, Y 8.6854, Z -2.1667, A 0.000, B 0.000, C 0.000 }
gfCNCPoint1[21154] = {X 482.0421, Y 8.2468, Z -2.1667, A 0.000, B 0.000, C 0.000 }
gfCNCPoint1[21155] = {X 484.1469, Y 7.9193, Z -2.1667, A 0.000, B 0.000, C 0.000 }
gfCNCPoint1[21156] = {X 486.2738, Y 7.8038, Z -2.1667, A 0.000, B 0.000, C 0.000 }
gfCNCPoint1[21157] = {X 486.9707, Y 7.7916, Z -2.1667, A 0.000, B 0.000, C 0.000 }
gfCNCPoint1[21158] = {X 502.2084, Y 7.7916, Z -2.1667, A 0.000, B 0.000, C 0.000 }
gfCNCPoint1[21159] = {X 502.7380, Y 7.7957, Z -2.1667, A 0.000, B 0.000, C 0.000 }
gfCNCPoint1[21160] = {X 503.7080, Y 7.9121, Z -2.1667, A 0.000, B 0.000, C 0.000 }
gfCNCPoint1[21161] = {X 504.6282, Y 8.2405, Z -2.1667, A 0.000, B 0.000, C 0.000 }
gfCNCPoint1[21162] = {X 505.4529, Y 8.7644, Z -2.1667, A 0.000, B 0.000, C 0.000 }
gfCNCPoint1[21163] = {X 506.1410, Y 9.4580, Z -2.1667, A 0.000, B 0.000, C 0.000 }
gfCNCPoint1[21164] = {X 506.6585, Y 10.2867, Z -2.1667, A 0.000, B 0.000, C 0.000 }
gfCNCPoint1[21165] = {X 506.9796, Y 11.2094, Z -2.1667, A 0.000, B 0.000, C 0.000 }
gfCNCPoint1[21166] = {X 507.0885, Y 12.1804, Z -2.1667, A 0.000, B 0.000, C 0.000 }
gfCNCPoint1[21167] = {X 507.0883, Y 13.0233, Z -2.1667, A 0.000, B 0.000, C 0.000 }
gfCNCPoint1[21168] = {X 506.9799, Y 13.9496, Z -2.1667, A 0.000, B 0.000, C 0.000 }
gfCNCPoint1[21169] = {X 506.6787, Y 14.8322, Z -2.1667, A 0.000, B 0.000, C 0.000 }
gfCNCPoint1[21170] = {X 506.1984, Y 15.6315, Z -2.1667, A 0.000, B 0.000, C 0.000 }
gfCNCPoint1[21171] = {X 505.5603, Y 16.3116, Z -2.1667, A 0.000, B 0.000, C 0.000 }
gfCNCPoint1[21172] = {X 505.5602, Y 40.8751, Z -2.1667, A 0.000, B 0.000, C 0.000 }
gfCNCPoint1[21173] = {X 506.2051, Y 41.5643, Z -2.1667, A 0.000, B 0.000, C 0.000 }
gfCNCPoint1[21174] = {X 506.6882, Y 42.3752, Z -2.1667, A 0.000, B 0.000, C 0.000 }
gfCNCPoint1[21175] = {X 506.9873, Y 43.2705, Z -2.1667, A 0.000, B 0.000, C 0.000 }
gfCNCPoint1[21176] = {X 507.0885, Y 44.2089, Z -2.1667, A 0.000, B 0.000, C 0.000 }
gfCNCPoint1[21177] = {X 507.0885, Y 45.0000, Z -2.1667, A 0.000, B 0.000, C 0.000 }
gfCNCPoint1[21178] = {X 506.9782, Y 45.9791, Z -2.1667, A 0.000, B 0.000, C 0.000 }
gfCNCPoint1[21179] = {X 506.6528, Y 46.9091, Z -2.1667, A 0.000, B 0.000, C 0.000 }
gfCNCPoint1[21180] = {X 506.1285, Y 47.7434, Z -2.1667, A 0.000, B 0.000, C 0.000 }
gfCNCPoint1[21181] = {X 505.4318, Y 48.4401, Z -2.1667, A 0.000, B 0.000, C 0.000 }
gfCNCPoint1[21182] = {X 504.5976, Y 48.9643, Z -2.1667, A 0.000, B 0.000, C 0.000 }
gfCNCPoint1[21183] = {X 503.6676, Y 49.2897, Z -2.1667, A 0.000, B 0.000, C 0.000 }
gfCNCPoint1[21184] = {X 502.6885, Y 49.4000, Z -2.1667, A 0.000, B 0.000, C 0.000 }
gfCNCPoint1[21185] = {X 496.2450, Y 49.4000, Z -2.1667, A 0.000, B 0.000, C 0.000 }
gfCNCPoint1[21186] = {X 495.2659, Y 49.2897, Z -2.1667, A 0.000, B 0.000, C 0.000 }
gfCNCPoint1[21187] = {X 494.3359, Y 48.9643, Z -2.1667, A 0.000, B 0.000, C 0.000 }
gfCNCPoint1[21188] = {X 493.5017, Y 48.4400, Z -2.1667, A 0.000, B 0.000, C 0.000 }
gfCNCPoint1[21189] = {X 492.8050, Y 47.7433, Z -2.1667, A 0.000, B 0.000, C 0.000 }
gfCNCPoint1[21190] = {X 492.2807, Y 46.9091, Z -2.1667, A 0.000, B 0.000, C 0.000 }
gfCNCPoint1[21191] = {X 491.9553, Y 45.9791, Z -2.1667, A 0.000, B 0.000, C 0.000 }
gfCNCPoint1[21192] = {X 491.8450, Y 45.0000, Z -2.1667, A 0.000, B 0.000, C 0.000 }
gfCNCPoint1[21193] = {X 491.8454, Y 44.1483, Z -2.1667, A 0.000, B 0.000, C 0.000 }
gfCNCPoint1[21194] = {X 491.9559, Y 43.2275, Z -2.1667, A 0.000, B 0.000, C 0.000 }
gfCNCPoint1[21195] = {X 492.2568, Y 42.3503, Z -2.1667, A 0.000, B 0.000, C 0.000 }
gfCNCPoint1[21196] = {X 492.7349, Y 41.5556, Z -2.1667, A 0.000, B 0.000, C 0.000 }
gfCNCPoint1[21197] = {X 493.3690, Y 40.8789, Z -2.1667, A 0.000, B 0.000, C 0.000 }
gfCNCPoint1[21198] = {X 493.3690, Y 34.5538, Z -2.1667, A 0.000, B 0.000, C 0.000 }
gfCNCPoint1[21199] = {X 490.7723, Y 34.5538, Z -2.1667, A 0.000, B 0.000, C 0.000 }
gfCNCPoint1[21200] = {X 486.5266, Y 42.8215, Z -2.1667, A 0.000, B 0.000, C 0.000 }
gfCNCPoint1[21201] = {X 486.6946, Y 43.5062, Z -2.1667, A 0.000, B 0.000, C 0.000 }
gfCNCPoint1[21202] = {X 486.7510, Y 44.2089, Z -2.1667, A 0.000, B 0.000, C 0.000 }
gfCNCPoint1[21203] = {X 486.7510, Y 45.0000, Z -2.1667, A 0.000, B 0.000, C 0.000 }
gfCNCPoint1[21204] = {X 486.6407, Y 45.9791, Z -2.1667, A 0.000, B 0.000, C 0.000 }
gfCNCPoint1[21205] = {X 486.3153, Y 46.9091, Z -2.1667, A 0.000, B 0.000, C 0.000 }
gfCNCPoint1[21206] = {X 485.7911, Y 47.7434, Z -2.1667, A 0.000, B 0.000, C 0.000 }
gfCNCPoint1[21207] = {X 485.0944, Y 48.4401, Z -2.1667, A 0.000, B 0.000, C 0.000 }
gfCNCPoint1[21208] = {X 484.2601, Y 48.9643, Z -2.1667, A 0.000, B 0.000, C 0.000 }
gfCNCPoint1[21209] = {X 483.3301, Y 49.2897, Z -2.1667, A 0.000, B 0.000, C 0.000 }
gfCNCPoint1[21210] = {X 482.3510, Y 49.4000, Z -2.1667, A 0.000, B 0.000, C 0.000 }
gfCNCPoint1[21211] = {X 480.2695, Y 49.4000, Z -2.1667, A 0.000, B 0.000, C 0.000 }
gfCNCPoint1[21212] = {X 480.2695, Y 49.8800, Z -2.1667, A 0.000, B 0.000, C 0.000 }
gfCNCPoint1[21213] = {X 481.4067, Y 50.7435, Z -2.1667, A 0.000, B 0.000, C 0.000 }
gfCNCPoint1[21214] = {X 482.4044, Y 51.7649, Z -2.1667, A 0.000, B 0.000, C 0.000 }
gfCNCPoint1[21215] = {X 483.2411, Y 52.9219, Z -2.1667, A 0.000, B 0.000, C 0.000 }
gfCNCPoint1[21216] = {X 483.8615, Y 54.1044, Z -2.1667, A 0.000, B 0.000, C 0.000 }
gfCNCPoint1[21217] = {X 484.3133, Y 55.3610, Z -2.1667, A 0.000, B 0.000, C 0.000 }
gfCNCPoint1[21218] = {X 484.5879, Y 56.6678, Z -2.1667, A 0.000, B 0.000, C 0.000 }
gfCNCPoint1[21219] = {X 484.6800, Y 58.0000, Z -2.1667, A 0.000, B 0.000, C 0.000 }
gfCNCPoint1[21220] = {X 484.6797, Y 59.0140, Z -2.1667, A 0.000, B 0.000, C 0.000 }
gfCNCPoint1[21221] = {X 484.5592, Y 60.4586, Z -2.1667, A 0.000, B 0.000, C 0.000 }
gfCNCPoint1[21222] = {X 484.2244, Y 61.8689, Z -2.1667, A 0.000, B 0.000, C 0.000 }
gfCNCPoint1[21223] = {X 483.6827, Y 63.2135, Z -2.1667, A 0.000, B 0.000, C 0.000 }
gfCNCPoint1[21224] = {X 482.9463, Y 64.4620, Z -2.1667, A 0.000, B 0.000, C 0.000 }
gfCNCPoint1[21225] = {X 482.0318, Y 65.5866, Z -2.1667, A 0.000, B 0.000, C 0.000 }
gfCNCPoint1[21226] = {X 480.9595, Y 66.5621, Z -2.1667, A 0.000, B 0.000, C 0.000 }
gfCNCPoint1[21227] = {X 480.9598, Y 89.4450, Z -2.1667, A 0.000, B 0.000, C 0.000 }
gfCNCPoint1[21228] = {X 482.0594, Y 90.4471, Z -2.1667, A 0.000, B 0.000, C 0.000 }
gfCNCPoint1[21229] = {X 482.9919, Y 91.6063, Z -2.1667, A 0.000, B 0.000, C 0.000 }
gfCNCPoint1[21230] = {X 483.7353, Y 92.8949, Z -2.1667, A 0.000, B 0.000, C 0.000 }
gfCNCPoint1[21231] = {X 507.6819, Y 92.8949, Z -2.1667, A 0.000, B 0.000, C 0.000 }
gfCNCPoint1[21232] = {X 507.6819, Y 95.2949, Z -2.1667, A 0.000, B 0.000, C 0.000 }
gfCNCPoint1[21233] = {X 595.2965, Y 95.2949, Z -2.1667, A 0.000, B 0.000, C 0.000 }
gfCNCPoint1[21234] = {X 595.2965, Y 54.2000, Z -2.1667, A 0.000, B 0.000, C 0.000 }
gfCNCPoint1[21235] = {X 593.5565, Y 54.2000, Z -2.1667, A 0.000, B 0.000, C 0.000 }
gfCNCPoint1[21236] = {X 592.2403, Y 54.1053, Z -2.1667, A 0.000, B 0.000, C 0.000 }
gfCNCPoint1[21237] = {X 590.9511, Y 53.8233, Z -2.1667, A 0.000, B 0.000, C 0.000 }
gfCNCPoint1[21238] = {X 589.7155, Y 53.3598, Z -2.1667, A 0.000, B 0.000, C 0.000 }
gfCNCPoint1[21239] = {X 588.5589, Y 52.7242, Z -2.1667, A 0.000, B 0.000, C 0.000 }
gfCNCPoint1[21240] = {X 587.5052, Y 51.9297, Z -2.1667, A 0.000, B 0.000, C 0.000 }
gfCNCPoint1[21241] = {X 586.4956, Y 52.6955, Z -2.1667, A 0.000, B 0.000, C 0.000 }
gfCNCPoint1[21242] = {X 585.3903, Y 53.3153, Z -2.1667, A 0.000, B 0.000, C 0.000 }
gfCNCPoint1[21243] = {X 584.1375, Y 53.7999, Z -2.1667, A 0.000, B 0.000, C 0.000 }
gfCNCPoint1[21244] = {X 582.8276, Y 54.0969, Z -2.1667, A 0.000, B 0.000, C 0.000 }
gfCNCPoint1[21245] = {X 581.4884, Y 54.1999, Z -2.1667, A 0.000, B 0.000, C 0.000 }
gfCNCPoint1[21246] = {X 580.1485, Y 54.1069, Z -2.1667, A 0.000, B 0.000, C 0.000 }
gfCNCPoint1[21247] = {X 578.8364, Y 53.8198, Z -2.1667, A 0.000, B 0.000, C 0.000 }
gfCNCPoint1[21248] = {X 577.5801, Y 53.3447, Z -2.1667, A 0.000, B 0.000, C 0.000 }
gfCNCPoint1[21249] = {X 576.4063, Y 52.6917, Z -2.1667, A 0.000, B 0.000, C 0.000 }
gfCNCPoint1[21250] = {X 575.3401, Y 51.8748, Z -2.1667, A 0.000, B 0.000, C 0.000 }
gfCNCPoint1[21251] = {X 574.2798, Y 52.6879, Z -2.1667, A 0.000, B 0.000, C 0.000 }
gfCNCPoint1[21252] = {X 573.1128, Y 53.3388, Z -2.1667, A 0.000, B 0.000, C 0.000 }
gfCNCPoint1[21253] = {X 571.8638, Y 53.8139, Z -2.1667, A 0.000, B 0.000, C 0.000 }
gfCNCPoint1[21254] = {X 570.5592, Y 54.1030, Z -2.1667, A 0.000, B 0.000, C 0.000 }
gfCNCPoint1[21255] = {X 569.2264, Y 54.2000, Z -2.1667, A 0.000, B 0.000, C 0.000 }
gfCNCPoint1[21256] = {X 562.4443, Y 54.2000, Z -2.1667, A 0.000, B 0.000, C 0.000 }
gfCNCPoint1[21257] = {X 561.0051, Y 54.0867, Z -2.1667, A 0.000, B 0.000, C 0.000 }
gfCNCPoint1[21258] = {X 559.6013, Y 53.7497, Z -2.1667, A 0.000, B 0.000, C 0.000 }
gfCNCPoint1[21259] = {X 558.2676, Y 53.1973, Z -2.1667, A 0.000, B 0.000, C 0.000 }
gfCNCPoint1[21260] = {X 557.0367, Y 52.4430, Z -2.1667, A 0.000, B 0.000, C 0.000 }
gfCNCPoint1[21261] = {X 555.9389, Y 51.5054, Z -2.1667, A 0.000, B 0.000, C 0.000 }
gfCNCPoint1[21262] = {X 555.0013, Y 50.4076, Z -2.1667, A 0.000, B 0.000, C 0.000 }
gfCNCPoint1[21263] = {X 554.2470, Y 49.1767, Z -2.1667, A 0.000, B 0.000, C 0.000 }
gfCNCPoint1[21264] = {X 553.6946, Y 47.8430, Z -2.1667, A 0.000, B 0.000, C 0.000 }
gfCNCPoint1[21265] = {X 553.3576, Y 46.4392, Z -2.1667, A 0.000, B 0.000, C 0.000 }
gfCNCPoint1[21266] = {X 553.2443, Y 45.0000, Z -2.1667, A 0.000, B 0.000, C 0.000 }
gfCNCPoint1[21267] = {X 553.2443, Y 44.0593, Z -2.1667, A 0.000, B 0.000, C 0.000 }
gfCNCPoint1[21268] = {X 553.3453, Y 42.7234, Z -2.1667, A 0.000, B 0.000, C 0.000 }
gfCNCPoint1[21269] = {X 553.6384, Y 41.4160, Z -2.1667, A 0.000, B 0.000, C 0.000 }
gfCNCPoint1[21270] = {X 554.1176, Y 40.1649, Z -2.1667, A 0.000, B 0.000, C 0.000 }
gfCNCPoint1[21271] = {X 554.7727, Y 38.9962, Z -2.1667, A 0.000, B 0.000, C 0.000 }
gfCNCPoint1[21272] = {X 554.7727, Y 11.0121, Z -2.1667, A 0.000, B 0.000, C 0.000 }
gfCNCPoint1[21273] = {X 554.1223, Y 9.8565, Z -2.1667, A 0.000, B 0.000, C 0.000 }
gfCNCPoint1[21274] = {X 553.6449, Y 8.6193, Z -2.1667, A 0.000, B 0.000, C 0.000 }
gfCNCPoint1[21275] = {X 553.3503, Y 7.3264, Z -2.1667, A 0.000, B 0.000, C 0.000 }
gfCNCPoint1[21276] = {X 553.2446, Y 6.0046, Z -2.1667, A 0.000, B 0.000, C 0.000 }
gfCNCPoint1[21277] = {X 553.2443, Y 5.0000, Z -2.1667, A 0.000, B 0.000, C 0.000 }
gfCNCPoint1[21278] = {X 553.2455, Y 4.8525, Z -2.1667, A 0.000, B 0.000, C 0.000 }
gfCNCPoint1[21279] = {X 553.2490, Y 4.7051, Z -2.1667, A 0.000, B 0.000, C 0.000 }
gfCNCPoint1[21280] = {X 365.1861, Y 4.7051, Z -2.1667, A 0.000, B 0.000, C 0.000 }
gfCNCPoint1[21281] = {X 365.5697, Y 5.1224, Z -2.1667, A 0.000, B 0.000, C 0.000 }
gfCNCPoint1[21282] = {X 365.9433, Y 5.5487, Z -2.1667, A 0.000, B 0.000, C 0.000 }
gfCNCPoint1[21283] = {X 367.0641, Y 6.9479, Z -2.1667, A 0.000, B 0.000, C 0.000 }
gfCNCPoint1[21284] = {X 368.0920, Y 8.4167, Z -2.1667, A 0.000, B 0.000, C 0.000 }
gfCNCPoint1[21285] = {X 369.3435, Y 10.5344, Z -2.1667, A 0.000, B 0.000, C 0.000 }
gfCNCPoint1[21286] = {X 370.4020, Y 12.7549, Z -2.1667, A 0.000, B 0.000, C 0.000 }
gfCNCPoint1[21287] = {X 371.2592, Y 15.0605, Z -2.1667, A 0.000, B 0.000, C 0.000 }
gfCNCPoint1[21288] = {X 371.9084, Y 17.4332, Z -2.1667, A 0.000, B 0.000, C 0.000 }
gfCNCPoint1[21289] = {X 372.3626, Y 19.8295, Z -2.1667, A 0.000, B 0.000, C 0.000 }
gfCNCPoint1[21290] = {X 372.6469, Y 22.2518, Z -2.1667, A 0.000, B 0.000, C 0.000 }
gfCNCPoint1[21291] = {X 372.7598, Y 24.6882, Z -2.1667, A 0.000, B 0.000, C 0.000 }
gfCNCPoint1[21292] = {X 372.7008, Y 27.1264, Z -2.1667, A 0.000, B 0.000, C 0.000 }
gfCNCPoint1[21293] = {X 372.4700, Y 29.5545, Z -2.1667, A 0.000, B 0.000, C 0.000 }
gfCNCPoint1[21294] = {X 372.0688, Y 31.9602, Z -2.1667, A 0.000, B 0.000, C 0.000 }
gfCNCPoint1[21295] = {X 371.4820, Y 34.3173, Z -2.1667, A 0.000, B 0.000, C 0.000 }
gfCNCPoint1[21296] = {X 370.6893, Y 36.6133, Z -2.1667, A 0.000, B 0.000, C 0.000 }
gfCNCPoint1[21297] = {X 369.6970, Y 38.8303, Z -2.1667, A 0.000, B 0.000, C 0.000 }
gfCNCPoint1[21298] = {X 368.5127, Y 40.9510, Z -2.1667, A 0.000, B 0.000, C 0.000 }
gfCNCPoint1[21299] = {X 367.1457, Y 42.9588, Z -2.1667, A 0.000, B 0.000, C 0.000 }
gfCNCPoint1[21300] = {X 365.7527, Y 44.6742, Z -2.1667, A 0.000, B 0.000, C 0.000 }
gfCNCPoint1[21301] = {X 364.2145, Y 46.2608, Z -2.1667, A 0.000, B 0.000, C 0.000 }
gfCNCPoint1[21302] = {X 362.5429, Y 47.7061, Z -2.1667, A 0.000, B 0.000, C 0.000 }
gfCNCPoint1[21303] = {X 360.7509, Y 48.9990, Z -2.1667, A 0.000, B 0.000, C 0.000 }
gfCNCPoint1[21304] = {X 358.8523, Y 50.1296, Z -2.1667, A 0.000, B 0.000, C 0.000 }
gfCNCPoint1[21305] = {X 356.6374, Y 51.1397, Z -2.1667, A 0.000, B 0.000, C 0.000 }
gfCNCPoint1[21306] = {X 354.3365, Y 51.9347, Z -2.1667, A 0.000, B 0.000, C 0.000 }
gfCNCPoint1[21307] = {X 351.9706, Y 52.5076, Z -2.1667, A 0.000, B 0.000, C 0.000 }
gfCNCPoint1[21308] = {X 349.5609, Y 52.8530, Z -2.1667, A 0.000, B 0.000, C 0.000 }
gfCNCPoint1[21309] = {X 347.1293, Y 52.9680, Z -2.1667, A 0.000, B 0.000, C 0.000 }
gfCNCPoint1[21310] = {X 344.8095, Y 52.9253, Z -2.1667, A 0.000, B 0.000, C 0.000 }
gfCNCPoint1[21311] = {X 342.5021, Y 52.6820, Z -2.1667, A 0.000, B 0.000, C 0.000 }
gfCNCPoint1[21312] = {X 340.2245, Y 52.2397, Z -2.1667, A 0.000, B 0.000, C 0.000 }
gfCNCPoint1[21313] = {X 337.9937, Y 51.6019, Z -2.1667, A 0.000, B 0.000, C 0.000 }
gfCNCPoint1[21314] = {X 335.8265, Y 50.7733, Z -2.1667, A 0.000, B 0.000, C 0.000 }
gfCNCPoint1[21315] = {X 333.7393, Y 49.7601, Z -2.1667, A 0.000, B 0.000, C 0.000 }
gfCNCPoint1[21316] = {X 332.8283, Y 49.2226, Z -2.1667, A 0.000, B 0.000, C 0.000 }
gfCNCPoint1[21317] = {X 331.9390, Y 48.6499, Z -2.1667, A 0.000, B 0.000, C 0.000 }
gfCNCPoint1[21318] = {X 331.3043, Y 48.2100, Z -2.1667, A 0.000, B 0.000, C 0.000 }
gfCNCPoint1[21319] = {X 330.6824, Y 47.7522, Z -2.1667, A 0.000, B 0.000, C 0.000 }
gfCNCPoint1[21320] = {X 329.2321, Y 49.6644, Z -2.1667, A 0.000, B 0.000, C 0.000 }
gfCNCPoint1[21321] = {X 328.8816, Y 49.3944, Z -2.1667, A 0.000, B 0.000, C 0.000 }
gfCNCPoint1[21322] = {X 328.5352, Y 49.1192, Z -2.1667, A 0.000, B 0.000, C 0.000 }
gfCNCPoint1[21323] = {X 328.1284, Y 49.0394, Z -2.1667, A 0.000, B 0.000, C 0.000 }
gfCNCPoint1[21324] = {X 327.7253, Y 48.9423, Z -2.1667, A 0.000, B 0.000, C 0.000 }
gfCNCPoint1[21325] = {X 328.4943, Y 49.2708, Z -2.1667, A 0.000, B 0.000, C 0.000 }
gfCNCPoint1[21326] = {X 329.2321, Y 49.6644, Z -2.1667, A 0.000, B 0.000, C 0.000 }
gfCNCPoint1[21327] = {X 330.6824, Y 47.7522, Z -2.1667, A 0.000, B 0.000, C 0.000 }
gfCNCPoint1[21328] = {X 330.1030, Y 47.3002, Z -2.1667, A 0.000, B 0.000, C 0.000 }
gfCNCPoint1[21329] = {X 329.5360, Y 46.8326, Z -2.1667, A 0.000, B 0.000, C 0.000 }
gfCNCPoint1[21330] = {X 328.9323, Y 46.7522, Z -2.1667, A 0.000, B 0.000, C 0.000 }
gfCNCPoint1[21331] = {X 328.3374, Y 46.6216, Z -2.1667, A 0.000, B 0.000, C 0.000 }
gfCNCPoint1[21332] = {X 327.9789, Y 46.5172, Z -2.1667, A 0.000, B 0.000, C 0.000 }
gfCNCPoint1[21333] = {X 327.6263, Y 46.3944, Z -2.1667, A 0.000, B 0.000, C 0.000 }
gfCNCPoint1[21334] = {X 326.7320, Y 45.9864, Z -2.1667, A 0.000, B 0.000, C 0.000 }
gfCNCPoint1[21335] = {X 325.9009, Y 45.4616, Z -2.1667, A 0.000, B 0.000, C 0.000 }
gfCNCPoint1[21336] = {X 325.1480, Y 44.8296, Z -2.1667, A 0.000, B 0.000, C 0.000 }
gfCNCPoint1[21337] = {X 324.5140, Y 44.2115, Z -2.1667, A 0.000, B 0.000, C 0.000 }
gfCNCPoint1[21338] = {X 324.0475, Y 43.7117, Z -2.1667, A 0.000, B 0.000, C 0.000 }
gfCNCPoint1[21339] = {X 323.6300, Y 43.1703, Z -2.1667, A 0.000, B 0.000, C 0.000 }
gfCNCPoint1[21340] = {X 319.6957, Y 45.9200, Z -2.1667, A 0.000, B 0.000, C 0.000 }
gfCNCPoint1[21341] = {X 319.4780, Y 45.5976, Z -2.1667, A 0.000, B 0.000, C 0.000 }
gfCNCPoint1[21342] = {X 319.2708, Y 45.2683, Z -2.1667, A 0.000, B 0.000, C 0.000 }
gfCNCPoint1[21343] = {X 319.2514, Y 45.5948, Z -2.1667, A 0.000, B 0.000, C 0.000 }
gfCNCPoint1[21344] = {X 319.2174, Y 45.9200, Z -2.1667, A 0.000, B 0.000, C 0.000 }
gfCNCPoint1[21345] = {X 319.6957, Y 45.9200, Z -2.1667, A 0.000, B 0.000, C 0.000 }
gfCNCPoint1[21346] = {X 321.6628, Y 44.5452, Z -2.1667, A 0.000, B 0.000, C 0.000 }
gfCNCPoint1[21347] = {X 321.4884, Y 44.2868, Z -2.1667, A 0.000, B 0.000, C 0.000 }
gfCNCPoint1[21348] = {X 321.3224, Y 44.0230, Z -2.1667, A 0.000, B 0.000, C 0.000 }
gfCNCPoint1[21349] = {X 320.6714, Y 42.7460, Z -2.1667, A 0.000, B 0.000, C 0.000 }
gfCNCPoint1[21350] = {X 320.2161, Y 41.3869, Z -2.1667, A 0.000, B 0.000, C 0.000 }
gfCNCPoint1[21351] = {X 319.9664, Y 39.9754, Z -2.1667, A 0.000, B 0.000, C 0.000 }
gfCNCPoint1[21352] = {X 319.9280, Y 38.5426, Z -2.1667, A 0.000, B 0.000, C 0.000 }
gfCNCPoint1[21353] = {X 320.1015, Y 37.1198, Z -2.1667, A 0.000, B 0.000, C 0.000 }
gfCNCPoint1[21354] = {X 320.4295, Y 35.8925, Z -2.1667, A 0.000, B 0.000, C 0.000 }
gfCNCPoint1[21355] = {X 320.9154, Y 34.7187, Z -2.1667, A 0.000, B 0.000, C 0.000 }
gfCNCPoint1[21356] = {X 321.5508, Y 33.6186, Z -2.1667, A 0.000, B 0.000, C 0.000 }
gfCNCPoint1[21357] = {X 324.1372, Y 29.7514, Z -2.1667, A 0.000, B 0.000, C 0.000 }
gfCNCPoint1[21358] = {X 320.1473, Y 27.0830, Z -2.1667, A 0.000, B 0.000, C 0.000 }
gfCNCPoint1[21359] = {X 321.8042, Y 24.6056, Z -2.1667, A 0.000, B 0.000, C 0.000 }
gfCNCPoint1[21360] = {X 321.9898, Y 24.3355, Z -2.1667, A 0.000, B 0.000, C 0.000 }
gfCNCPoint1[21361] = {X 322.1814, Y 24.0697, Z -2.1667, A 0.000, B 0.000, C 0.000 }
gfCNCPoint1[21362] = {X 321.5380, Y 23.0772, Z -2.1667, A 0.000, B 0.000, C 0.000 }
gfCNCPoint1[21363] = {X 320.9777, Y 22.0354, Z -2.1667, A 0.000, B 0.000, C 0.000 }
gfCNCPoint1[21364] = {X 320.1474, Y 20.3274, Z -2.1667, A 0.000, B 0.000, C 0.000 }
gfCNCPoint1[21365] = {X 320.1473, Y 27.0830, Z -2.1667, A 0.000, B 0.000, C 0.000 }
gfCNCPoint1[21366] = {X 322.1423, Y 28.4172, Z -2.1667, A 0.000, B 0.000, C 0.000 }
gfCNCPoint1[21367] = {X 323.7975, Y 25.9423, Z -2.1667, A 0.000, B 0.000, C 0.000 }
gfCNCPoint1[21368] = {X 324.5112, Y 24.9841, Z -2.1667, A 0.000, B 0.000, C 0.000 }
gfCNCPoint1[21369] = {X 325.3162, Y 24.1010, Z -2.1667, A 0.000, B 0.000, C 0.000 }
gfCNCPoint1[21370] = {X 324.4812, Y 23.1413, Z -2.1667, A 0.000, B 0.000, C 0.000 }
gfCNCPoint1[21371] = {X 323.7518, Y 22.0991, Z -2.1667, A 0.000, B 0.000, C 0.000 }
gfCNCPoint1[21372] = {X 323.1360, Y 20.9859, Z -2.1667, A 0.000, B 0.000, C 0.000 }
gfCNCPoint1[21373] = {X 319.6151, Y 13.7428, Z -2.1667, A 0.000, B 0.000, C 0.000 }
gfCNCPoint1[21374] = {X 319.4387, Y 13.3633, Z -2.1667, A 0.000, B 0.000, C 0.000 }
gfCNCPoint1[21375] = {X 319.2755, Y 12.9779, Z -2.1667, A 0.000, B 0.000, C 0.000 }
gfCNCPoint1[21376] = {X 319.2755, Y 13.0353, Z -2.1667, A 0.000, B 0.000, C 0.000 }
gfCNCPoint1[21377] = {X 319.1697, Y 14.2159, Z -2.1667, A 0.000, B 0.000, C 0.000 }
gfCNCPoint1[21378] = {X 318.8737, Y 15.3637, Z -2.1667, A 0.000, B 0.000, C 0.000 }
gfCNCPoint1[21379] = {X 318.3954, Y 16.4482, Z -2.1667, A 0.000, B 0.000, C 0.000 }
gfCNCPoint1[21380] = {X 317.7474, Y 17.4408, Z -2.1667, A 0.000, B 0.000, C 0.000 }
gfCNCPoint1[21381] = {X 317.7472, Y 36.6537, Z -2.1667, A 0.000, B 0.000, C 0.000 }
gfCNCPoint1[21382] = {X 318.1565, Y 35.1220, Z -2.1667, A 0.000, B 0.000, C 0.000 }
gfCNCPoint1[21383] = {X 318.7629, Y 33.6572, Z -2.1667, A 0.000, B 0.000, C 0.000 }
gfCNCPoint1[21384] = {X 319.5559, Y 32.2844, Z -2.1667, A 0.000, B 0.000, C 0.000 }
gfCNCPoint1[21385] = {X 322.1423, Y 28.4172, Z -2.1667, A 0.000, B 0.000, C 0.000 }
gfCNCPoint1[21386] = {X 324.1372, Y 29.7514, Z -2.1667, A 0.000, B 0.000, C 0.000 }
gfCNCPoint1[21387] = {X 325.7908, Y 27.2790, Z -2.1667, A 0.000, B 0.000, C 0.000 }
gfCNCPoint1[21388] = {X 326.3627, Y 26.5111, Z -2.1667, A 0.000, B 0.000, C 0.000 }
gfCNCPoint1[21389] = {X 327.0077, Y 25.8035, Z -2.1667, A 0.000, B 0.000, C 0.000 }
gfCNCPoint1[21390] = {X 328.0707, Y 24.8904, Z -2.1667, A 0.000, B 0.000, C 0.000 }
gfCNCPoint1[21391] = {X 329.2543, Y 24.1403, Z -2.1667, A 0.000, B 0.000, C 0.000 }
gfCNCPoint1[21392] = {X 328.0859, Y 23.3667, Z -2.1667, A 0.000, B 0.000, C 0.000 }
gfCNCPoint1[21393] = {X 327.0414, Y 22.4326, Z -2.1667, A 0.000, B 0.000, C 0.000 }
gfCNCPoint1[21394] = {X 326.3723, Y 21.6635, Z -2.1667, A 0.000, B 0.000, C 0.000 }
gfCNCPoint1[21395] = {X 325.7878, Y 20.8284, Z -2.1667, A 0.000, B 0.000, C 0.000 }
gfCNCPoint1[21396] = {X 325.2944, Y 19.9364, Z -2.1667, A 0.000, B 0.000, C 0.000 }
gfCNCPoint1[21397] = {X 321.7736, Y 12.6936, Z -2.1667, A 0.000, B 0.000, C 0.000 }
gfCNCPoint1[21398] = {X 321.6322, Y 12.3894, Z -2.1667, A 0.000, B 0.000, C 0.000 }
gfCNCPoint1[21399] = {X 321.5015, Y 12.0806, Z -2.1667, A 0.000, B 0.000, C 0.000 }
gfCNCPoint1[21400] = {X 321.1058, Y 10.8774, Z -2.1667, A 0.000, B 0.000, C 0.000 }
gfCNCPoint1[21401] = {X 320.8706, Y 9.6328, Z -2.1667, A 0.000, B 0.000, C 0.000 }
gfCNCPoint1[21402] = {X 320.7999, Y 8.3681, Z -2.1667, A 0.000, B 0.000, C 0.000 }
gfCNCPoint1[21403] = {X 320.8950, Y 7.1051, Z -2.1667, A 0.000, B 0.000, C 0.000 }
gfCNCPoint1[21404] = {X 298.7842, Y 7.1051, Z -2.1667, A 0.000, B 0.000, C 0.000 }
gfCNCPoint1[21405] = {X 298.7842, Y 9.5051, Z -2.1667, A 0.000, B 0.000, C 0.000 }
gfCNCPoint1[21406] = {X 297.8292, Y 9.5051, Z -2.1667, A 0.000, B 0.000, C 0.000 }
gfCNCPoint1[21407] = {X 298.1372, Y 10.4756, Z -2.1667, A 0.000, B 0.000, C 0.000 }
gfCNCPoint1[21408] = {X 298.3067, Y 11.4795, Z -2.1667, A 0.000, B 0.000, C 0.000 }
gfCNCPoint1[21409] = {X 298.4762, Y 10.4756, Z -2.1667, A 0.000, B 0.000, C 0.000 }
gfCNCPoint1[21410] = {X 298.7842, Y 9.5051, Z -2.1667, A 0.000, B 0.000, C 0.000 }
gfCNCPoint1[21411] = {X 298.7842, Y 7.1051, Z -2.1667, A 0.000, B 0.000, C 0.000 }
gfCNCPoint1[21412] = {X 233.3052, Y 7.1051, Z -2.1667, A 0.000, B 0.000, C 0.000 }
gfCNCPoint1[21413] = {X 233.3052, Y 11.9051, Z -2.1667, A 0.000, B 0.000, C 0.000 }
gfCNCPoint1[21414] = {X 233.1564, Y 11.9051, Z -2.1667, A 0.000, B 0.000, C 0.000 }
gfCNCPoint1[21415] = {X 233.1595, Y 12.0458, Z -2.1667, A 0.000, B 0.000, C 0.000 }
gfCNCPoint1[21416] = {X 233.1605, Y 12.1866, Z -2.1667, A 0.000, B 0.000, C 0.000 }
gfCNCPoint1[21417] = {X 233.2322, Y 12.0455, Z -2.1667, A 0.000, B 0.000, C 0.000 }
gfCNCPoint1[21418] = {X 233.3052, Y 11.9051, Z -2.1667, A 0.000, B 0.000, C 0.000 }
gfCNCPoint1[21419] = {X 233.3052, Y 9.5051, Z -2.1667, A 0.000, B 0.000, C 0.000 }
gfCNCPoint1[21420] = {X 230.2485, Y 9.5051, Z -2.1667, A 0.000, B 0.000, C 0.000 }
gfCNCPoint1[21421] = {X 230.6107, Y 10.7178, Z -2.1667, A 0.000, B 0.000, C 0.000 }
gfCNCPoint1[21422] = {X 230.7574, Y 11.9749, Z -2.1667, A 0.000, B 0.000, C 0.000 }
gfCNCPoint1[21423] = {X 230.7597, Y 12.0809, Z -2.1667, A 0.000, B 0.000, C 0.000 }
gfCNCPoint1[21424] = {X 230.7605, Y 12.1868, Z -2.1667, A 0.000, B 0.000, C 0.000 }
gfCNCPoint1[21425] = {X 230.7602, Y 13.0462, Z -2.1667, A 0.000, B 0.000, C 0.000 }
gfCNCPoint1[21426] = {X 230.6531, Y 14.2239, Z -2.1667, A 0.000, B 0.000, C 0.000 }
gfCNCPoint1[21427] = {X 230.3567, Y 15.3687, Z -2.1667, A 0.000, B 0.000, C 0.000 }
gfCNCPoint1[21428] = {X 229.8790, Y 16.4504, Z -2.1667, A 0.000, B 0.000, C 0.000 }
gfCNCPoint1[21429] = {X 229.2324, Y 17.4405, Z -2.1667, A 0.000, B 0.000, C 0.000 }
gfCNCPoint1[21430] = {X 229.2327, Y 25.8423, Z -2.1667, A 0.000, B 0.000, C 0.000 }
gfCNCPoint1[21431] = {X 231.6327, Y 25.8422, Z -2.1667, A 0.000, B 0.000, C 0.000 }
gfCNCPoint1[21432] = {X 231.6332, Y 38.9900, Z -2.1667, A 0.000, B 0.000, C 0.000 }
gfCNCPoint1[21433] = {X 231.6440, Y 39.0069, Z -2.1667, A 0.000, B 0.000, C 0.000 }
gfCNCPoint1[21434] = {X 232.3931, Y 37.9855, Z -2.1667, A 0.000, B 0.000, C 0.000 }
gfCNCPoint1[21435] = {X 233.2692, Y 37.0706, Z -2.1667, A 0.000, B 0.000, C 0.000 }
gfCNCPoint1[21436] = {X 234.2573, Y 36.2780, Z -2.1667, A 0.000, B 0.000, C 0.000 }
gfCNCPoint1[21437] = {X 235.5697, Y 33.7091, Z -2.1667, A 0.000, B 0.000, C 0.000 }
gfCNCPoint1[21438] = {X 234.4291, Y 32.2850, Z -2.1667, A 0.000, B 0.000, C 0.000 }
gfCNCPoint1[21439] = {X 233.4509, Y 30.7448, Z -2.1667, A 0.000, B 0.000, C 0.000 }
gfCNCPoint1[21440] = {X 232.6469, Y 29.1070, Z -2.1667, A 0.000, B 0.000, C 0.000 }
gfCNCPoint1[21441] = {X 232.0265, Y 27.3912, Z -2.1667, A 0.000, B 0.000, C 0.000 }
gfCNCPoint1[21442] = {X 231.8155, Y 26.6203, Z -2.1667, A 0.000, B 0.000, C 0.000 }
gfCNCPoint1[21443] = {X 231.6327, Y 25.8422, Z -2.1667, A 0.000, B 0.000, C 0.000 }
gfCNCPoint1[21444] = {X 229.2327, Y 25.8423, Z -2.1667, A 0.000, B 0.000, C 0.000 }
gfCNCPoint1[21445] = {X 229.2332, Y 39.7473, Z -2.1667, A 0.000, B 0.000, C 0.000 }
gfCNCPoint1[21446] = {X 229.4329, Y 40.0175, Z -2.1667, A 0.000, B 0.000, C 0.000 }
gfCNCPoint1[21447] = {X 229.6200, Y 40.2966, Z -2.1667, A 0.000, B 0.000, C 0.000 }
gfCNCPoint1[21448] = {X 230.1055, Y 41.1910, Z -2.1667, A 0.000, B 0.000, C 0.000 }
gfCNCPoint1[21449] = {X 230.4616, Y 42.1443, Z -2.1667, A 0.000, B 0.000, C 0.000 }
gfCNCPoint1[21450] = {X 230.6813, Y 43.1379, Z -2.1667, A 0.000, B 0.000, C 0.000 }
gfCNCPoint1[21451] = {X 230.7603, Y 44.1524, Z -2.1667, A 0.000, B 0.000, C 0.000 }
gfCNCPoint1[21452] = {X 230.7605, Y 45.0000, Z -2.1667, A 0.000, B 0.000, C 0.000 }
gfCNCPoint1[21453] = {X 230.7459, Y 45.4609, Z -2.1667, A 0.000, B 0.000, C 0.000 }
gfCNCPoint1[21454] = {X 230.7021, Y 45.9200, Z -2.1667, A 0.000, B 0.000, C 0.000 }
gfCNCPoint1[21455] = {X 232.5859, Y 45.9200, Z -2.1667, A 0.000, B 0.000, C 0.000 }
gfCNCPoint1[21456] = {X 232.5421, Y 45.4609, Z -2.1667, A 0.000, B 0.000, C 0.000 }
gfCNCPoint1[21457] = {X 232.5275, Y 45.0000, Z -2.1667, A 0.000, B 0.000, C 0.000 }
gfCNCPoint1[21458] = {X 232.5275, Y 44.2090, Z -2.1667, A 0.000, B 0.000, C 0.000 }
gfCNCPoint1[21459] = {X 232.6006, Y 43.1799, Z -2.1667, A 0.000, B 0.000, C 0.000 }
gfCNCPoint1[21460] = {X 232.8184, Y 42.1714, Z -2.1667, A 0.000, B 0.000, C 0.000 }
gfCNCPoint1[21461] = {X 233.1766, Y 41.2038, Z -2.1667, A 0.000, B 0.000, C 0.000 }
gfCNCPoint1[21462] = {X 233.6680, Y 40.2966, Z -2.1667, A 0.000, B 0.000, C 0.000 }
gfCNCPoint1[21463] = {X 234.3527, Y 39.3876, Z -2.1667, A 0.000, B 0.000, C 0.000 }
gfCNCPoint1[21464] = {X 235.1707, Y 38.5964, Z -2.1667, A 0.000, B 0.000, C 0.000 }
gfCNCPoint1[21465] = {X 236.1021, Y 37.9424, Z -2.1667, A 0.000, B 0.000, C 0.000 }
gfCNCPoint1[21466] = {X 238.5003, Y 33.2480, Z -2.1667, A 0.000, B 0.000, C 0.000 }
gfCNCPoint1[21467] = {X 237.3867, Y 32.1404, Z -2.1667, A 0.000, B 0.000, C 0.000 }
gfCNCPoint1[21468] = {X 236.4015, Y 30.9171, Z -2.1667, A 0.000, B 0.000, C 0.000 }
gfCNCPoint1[21469] = {X 235.5567, Y 29.5930, Z -2.1667, A 0.000, B 0.000, C 0.000 }
gfCNCPoint1[21470] = {X 234.8624, Y 28.1841, Z -2.1667, A 0.000, B 0.000, C 0.000 }
gfCNCPoint1[21471] = {X 234.3271, Y 26.7075, Z -2.1667, A 0.000, B 0.000, C 0.000 }
gfCNCPoint1[21472] = {X 234.1404, Y 26.0250, Z -2.1667, A 0.000, B 0.000, C 0.000 }
gfCNCPoint1[21473] = {X 233.9787, Y 25.3362, Z -2.1667, A 0.000, B 0.000, C 0.000 }
gfCNCPoint1[21474] = {X 233.6676, Y 23.4491, Z -2.1667, A 0.000, B 0.000, C 0.000 }
gfCNCPoint1[21475] = {X 233.5430, Y 21.5406, Z -2.1667, A 0.000, B 0.000, C 0.000 }
gfCNCPoint1[21476] = {X 233.6059, Y 19.6290, Z -2.1667, A 0.000, B 0.000, C 0.000 }
gfCNCPoint1[21477] = {X 233.8558, Y 17.7328, Z -2.1667, A 0.000, B 0.000, C 0.000 }
gfCNCPoint1[21478] = {X 234.2903, Y 15.8703, Z -2.1667, A 0.000, B 0.000, C 0.000 }
gfCNCPoint1[21479] = {X 234.7359, Y 14.5434, Z -2.1667, A 0.000, B 0.000, C 0.000 }
gfCNCPoint1[21480] = {X 235.3048, Y 13.2645, Z -2.1667, A 0.000, B 0.000, C 0.000 }
gfCNCPoint1[21481] = {X 235.3665, Y 13.1431, Z -2.1667, A 0.000, B 0.000, C 0.000 }
gfCNCPoint1[21482] = {X 235.4293, Y 13.0223, Z -2.1667, A 0.000, B 0.000, C 0.000 }
gfCNCPoint1[21483] = {X 236.1706, Y 11.7671, Z -2.1667, A 0.000, B 0.000, C 0.000 }
gfCNCPoint1[21484] = {X 237.0318, Y 10.5909, Z -2.1667, A 0.000, B 0.000, C 0.000 }
gfCNCPoint1[21485] = {X 238.0044, Y 9.5051, Z -2.1667, A 0.000, B 0.000, C 0.000 }
gfCNCPoint1[21486] = {X 233.3052, Y 9.5051, Z -2.1667, A 0.000, B 0.000, C 0.000 }
gfCNCPoint1[21487] = {X 233.3052, Y 7.1051, Z -2.1667, A 0.000, B 0.000, C 0.000 }
gfCNCPoint1[21488] = {X 207.3611, Y 7.1051, Z -2.1667, A 0.000, B 0.000, C 0.000 }
gfCNCPoint1[21489] = {X 207.3611, Y 11.9051, Z -2.1667, A 0.000, B 0.000, C 0.000 }
gfCNCPoint1[21490] = {X 205.8552, Y 11.9051, Z -2.1667, A 0.000, B 0.000, C 0.000 }
gfCNCPoint1[21491] = {X 206.6103, Y 13.3411, Z -2.1667, A 0.000, B 0.000, C 0.000 }
gfCNCPoint1[21492] = {X 207.2360, Y 14.8379, Z -2.1667, A 0.000, B 0.000, C 0.000 }
gfCNCPoint1[21493] = {X 207.7970, Y 16.7109, Z -2.1667, A 0.000, B 0.000, C 0.000 }
gfCNCPoint1[21494] = {X 208.1760, Y 18.6291, Z -2.1667, A 0.000, B 0.000, C 0.000 }
gfCNCPoint1[21495] = {X 208.3695, Y 20.5747, Z -2.1667, A 0.000, B 0.000, C 0.000 }
gfCNCPoint1[21496] = {X 208.3757, Y 22.5300, Z -2.1667, A 0.000, B 0.000, C 0.000 }
gfCNCPoint1[21497] = {X 208.1945, Y 24.4768, Z -2.1667, A 0.000, B 0.000, C 0.000 }
gfCNCPoint1[21498] = {X 207.8276, Y 26.3973, Z -2.1667, A 0.000, B 0.000, C 0.000 }
gfCNCPoint1[21499] = {X 207.3606, Y 28.0095, Z -2.1667, A 0.000, B 0.000, C 0.000 }
gfCNCPoint1[21500] = {X 206.7374, Y 29.5680, Z -2.1667, A 0.000, B 0.000, C 0.000 }
gfCNCPoint1[21501] = {X 205.9641, Y 31.0576, Z -2.1667, A 0.000, B 0.000, C 0.000 }
gfCNCPoint1[21502] = {X 206.0463, Y 31.2161, Z -2.1667, A 0.000, B 0.000, C 0.000 }
gfCNCPoint1[21503] = {X 206.1255, Y 31.3761, Z -2.1667, A 0.000, B 0.000, C 0.000 }
gfCNCPoint1[21504] = {X 208.8859, Y 37.0789, Z -2.1667, A 0.000, B 0.000, C 0.000 }
gfCNCPoint1[21505] = {X 208.8859, Y 18.1992, Z -2.1667, A 0.000, B 0.000, C 0.000 }
gfCNCPoint1[21506] = {X 208.2335, Y 17.0030, Z -2.1667, A 0.000, B 0.000, C 0.000 }
gfCNCPoint1[21507] = {X 207.7555, Y 15.7269, Z -2.1667, A 0.000, B 0.000, C 0.000 }
gfCNCPoint1[21508] = {X 207.4615, Y 14.3964, Z -2.1667, A 0.000, B 0.000, C 0.000 }
gfCNCPoint1[21509] = {X 207.3572, Y 13.0378, Z -2.1667, A 0.000, B 0.000, C 0.000 }
gfCNCPoint1[21510] = {X 207.3570, Y 12.1868, Z -2.1667, A 0.000, B 0.000, C 0.000 }
gfCNCPoint1[21511] = {X 207.3580, Y 12.0459, Z -2.1667, A 0.000, B 0.000, C 0.000 }
gfCNCPoint1[21512] = {X 207.3611, Y 11.9051, Z -2.1667, A 0.000, B 0.000, C 0.000 }
gfCNCPoint1[21513] = {X 207.3611, Y 9.5051, Z -2.1667, A 0.000, B 0.000, C 0.000 }
gfCNCPoint1[21514] = {X 200.9063, Y 9.5051, Z -2.1667, A 0.000, B 0.000, C 0.000 }
gfCNCPoint1[21515] = {X 201.9796, Y 10.6138, Z -2.1667, A 0.000, B 0.000, C 0.000 }
gfCNCPoint1[21516] = {X 202.9413, Y 11.8207, Z -2.1667, A 0.000, B 0.000, C 0.000 }
gfCNCPoint1[21517] = {X 203.7823, Y 13.1145, Z -2.1667, A 0.000, B 0.000, C 0.000 }
gfCNCPoint1[21518] = {X 204.4356, Y 14.3564, Z -2.1667, A 0.000, B 0.000, C 0.000 }
gfCNCPoint1[21519] = {X 204.9777, Y 15.6507, Z -2.1667, A 0.000, B 0.000, C 0.000 }
gfCNCPoint1[21520] = {X 205.5504, Y 17.6374, Z -2.1667, A 0.000, B 0.000, C 0.000 }
gfCNCPoint1[21521] = {X 205.8912, Y 19.6767, Z -2.1667, A 0.000, B 0.000, C 0.000 }
gfCNCPoint1[21522] = {X 205.9957, Y 21.7416, Z -2.1667, A 0.000, B 0.000, C 0.000 }
gfCNCPoint1[21523] = {X 205.8625, Y 23.8049, Z -2.1667, A 0.000, B 0.000, C 0.000 }
gfCNCPoint1[21524] = {X 205.4933, Y 25.8392, Z -2.1667, A 0.000, B 0.000, C 0.000 }
gfCNCPoint1[21525] = {X 205.0923, Y 27.2253, Z -2.1667, A 0.000, B 0.000, C 0.000 }
gfCNCPoint1[21526] = {X 204.5569, Y 28.5653, Z -2.1667, A 0.000, B 0.000, C 0.000 }
gfCNCPoint1[21527] = {X 203.8923, Y 29.8461, Z -2.1667, A 0.000, B 0.000, C 0.000 }
gfCNCPoint1[21528] = {X 203.1049, Y 31.0553, Z -2.1667, A 0.000, B 0.000, C 0.000 }
gfCNCPoint1[21529] = {X 203.5731, Y 31.7146, Z -2.1667, A 0.000, B 0.000, C 0.000 }
gfCNCPoint1[21530] = {X 203.9653, Y 32.4217, Z -2.1667, A 0.000, B 0.000, C 0.000 }
gfCNCPoint1[21531] = {X 206.9865, Y 38.6634, Z -2.1667, A 0.000, B 0.000, C 0.000 }
gfCNCPoint1[21532] = {X 207.4240, Y 39.8017, Z -2.1667, A 0.000, B 0.000, C 0.000 }
gfCNCPoint1[21533] = {X 207.6653, Y 40.9971, Z -2.1667, A 0.000, B 0.000, C 0.000 }
gfCNCPoint1[21534] = {X 207.7038, Y 42.2159, Z -2.1667, A 0.000, B 0.000, C 0.000 }
gfCNCPoint1[21535] = {X 207.5382, Y 43.4241, Z -2.1667, A 0.000, B 0.000, C 0.000 }
gfCNCPoint1[21536] = {X 207.1733, Y 44.5877, Z -2.1667, A 0.000, B 0.000, C 0.000 }
gfCNCPoint1[21537] = {X 206.6193, Y 45.6741, Z -2.1667, A 0.000, B 0.000, C 0.000 }
gfCNCPoint1[21538] = {X 205.8917, Y 46.6527, Z -2.1667, A 0.000, B 0.000, C 0.000 }
gfCNCPoint1[21539] = {X 205.0110, Y 47.4962, Z -2.1667, A 0.000, B 0.000, C 0.000 }
gfCNCPoint1[21540] = {X 204.4728, Y 47.9313, Z -2.1667, A 0.000, B 0.000, C 0.000 }
gfCNCPoint1[21541] = {X 203.5888, Y 48.5430, Z -2.1667, A 0.000, B 0.000, C 0.000 }
gfCNCPoint1[21542] = {X 202.6246, Y 49.0181, Z -2.1667, A 0.000, B 0.000, C 0.000 }
gfCNCPoint1[21543] = {X 201.4901, Y 49.3722, Z -2.1667, A 0.000, B 0.000, C 0.000 }
gfCNCPoint1[21544] = {X 200.3131, Y 49.5374, Z -2.1667, A 0.000, B 0.000, C 0.000 }
gfCNCPoint1[21545] = {X 199.1249, Y 49.5094, Z -2.1667, A 0.000, B 0.000, C 0.000 }
gfCNCPoint1[21546] = {X 196.8339, Y 50.6065, Z -2.1667, A 0.000, B 0.000, C 0.000 }
gfCNCPoint1[21547] = {X 194.4621, Y 51.5160, Z -2.1667, A 0.000, B 0.000, C 0.000 }
gfCNCPoint1[21548] = {X 192.0249, Y 52.2321, Z -2.1667, A 0.000, B 0.000, C 0.000 }
gfCNCPoint1[21549] = {X 190.7219, Y 52.5177, Z -2.1667, A 0.000, B 0.000, C 0.000 }
gfCNCPoint1[21550] = {X 189.4058, Y 52.7350, Z -2.1667, A 0.000, B 0.000, C 0.000 }
gfCNCPoint1[21551] = {X 189.9003, Y 53.9107, Z -2.1667, A 0.000, B 0.000, C 0.000 }
gfCNCPoint1[21552] = {X 190.2681, Y 55.1321, Z -2.1667, A 0.000, B 0.000, C 0.000 }
gfCNCPoint1[21553] = {X 190.5268, Y 56.5557, Z -2.1667, A 0.000, B 0.000, C 0.000 }
gfCNCPoint1[21554] = {X 190.6135, Y 58.0000, Z -2.1667, A 0.000, B 0.000, C 0.000 }
gfCNCPoint1[21555] = {X 190.6132, Y 58.8775, Z -2.1667, A 0.000, B 0.000, C 0.000 }
gfCNCPoint1[21556] = {X 208.6243, Y 78.5343, Z -2.1667, A 0.000, B 0.000, C 0.000 }
gfCNCPoint1[21557] = {X 212.1633, Y 75.2915, Z -2.1667, A 0.000, B 0.000, C 0.000 }
gfCNCPoint1[21558] = {X 215.1993, Y 78.6049, Z -2.1667, A 0.000, B 0.000, C 0.000 }
gfCNCPoint1[21559] = {X 218.3292, Y 76.5997, Z -2.1667, A 0.000, B 0.000, C 0.000 }
gfCNCPoint1[21560] = {X 216.9966, Y 76.0767, Z -2.1667, A 0.000, B 0.000, C 0.000 }
gfCNCPoint1[21561] = {X 216.3775, Y 75.8846, Z -2.1667, A 0.000, B 0.000, C 0.000 }
gfCNCPoint1[21562] = {X 215.7344, Y 75.8035, Z -2.1667, A 0.000, B 0.000, C 0.000 }
gfCNCPoint1[21563] = {X 213.9352, Y 75.6432, Z -2.1667, A 0.000, B 0.000, C 0.000 }
gfCNCPoint1[21564] = {X 212.1633, Y 75.2915, Z -2.1667, A 0.000, B 0.000, C 0.000 }
gfCNCPoint1[21565] = {X 210.3938, Y 76.9129, Z -2.1667, A 0.000, B 0.000, C 0.000 }
gfCNCPoint1[21566] = {X 214.7939, Y 81.7150, Z -2.1667, A 0.000, B 0.000, C 0.000 }
gfCNCPoint1[21567] = {X 223.5838, Y 76.0837, Z -2.1667, A 0.000, B 0.000, C 0.000 }
gfCNCPoint1[21568] = {X 217.8857, Y 73.8475, Z -2.1667, A 0.000, B 0.000, C 0.000 }
gfCNCPoint1[21569] = {X 216.8730, Y 73.5363, Z -2.1667, A 0.000, B 0.000, C 0.000 }
gfCNCPoint1[21570] = {X 215.8216, Y 73.4051, Z -2.1667, A 0.000, B 0.000, C 0.000 }
gfCNCPoint1[21571] = {X 214.2770, Y 73.2677, Z -2.1667, A 0.000, B 0.000, C 0.000 }
gfCNCPoint1[21572] = {X 212.7559, Y 72.9658, Z -2.1667, A 0.000, B 0.000, C 0.000 }
gfCNCPoint1[21573] = {X 211.1570, Y 72.4582, Z -2.1667, A 0.000, B 0.000, C 0.000 }
gfCNCPoint1[21574] = {X 209.6275, Y 71.7690, Z -2.1667, A 0.000, B 0.000, C 0.000 }
gfCNCPoint1[21575] = {X 208.1880, Y 70.9076, Z -2.1667, A 0.000, B 0.000, C 0.000 }
gfCNCPoint1[21576] = {X 206.8578, Y 69.8854, Z -2.1667, A 0.000, B 0.000, C 0.000 }
gfCNCPoint1[21577] = {X 205.6548, Y 68.7163, Z -2.1667, A 0.000, B 0.000, C 0.000 }
gfCNCPoint1[21578] = {X 204.5950, Y 67.4159, Z -2.1667, A 0.000, B 0.000, C 0.000 }
gfCNCPoint1[21579] = {X 203.6928, Y 66.0016, Z -2.1667, A 0.000, B 0.000, C 0.000 }
gfCNCPoint1[21580] = {X 202.9601, Y 64.4925, Z -2.1667, A 0.000, B 0.000, C 0.000 }
gfCNCPoint1[21581] = {X 202.4070, Y 62.9087, Z -2.1667, A 0.000, B 0.000, C 0.000 }
gfCNCPoint1[21582] = {X 202.0407, Y 61.2716, Z -2.1667, A 0.000, B 0.000, C 0.000 }
gfCNCPoint1[21583] = {X 199.6722, Y 61.6591, Z -2.1667, A 0.000, B 0.000, C 0.000 }
gfCNCPoint1[21584] = {X 199.5095, Y 60.3407, Z -2.1667, A 0.000, B 0.000, C 0.000 }
gfCNCPoint1[21585] = {X 199.4510, Y 59.0136, Z -2.1667, A 0.000, B 0.000, C 0.000 }
gfCNCPoint1[21586] = {X 199.4508, Y 58.0000, Z -2.1667, A 0.000, B 0.000, C 0.000 }
gfCNCPoint1[21587] = {X 199.5412, Y 56.2556, Z -2.1667, A 0.000, B 0.000, C 0.000 }
gfCNCPoint1[21588] = {X 199.8114, Y 54.5298, Z -2.1667, A 0.000, B 0.000, C 0.000 }
gfCNCPoint1[21589] = {X 197.5977, Y 55.4810, Z -2.1667, A 0.000, B 0.000, C 0.000 }
gfCNCPoint1[21590] = {X 195.3260, Y 56.2837, Z -2.1667, A 0.000, B 0.000, C 0.000 }
gfCNCPoint1[21591] = {X 195.3578, Y 56.6303, Z -2.1667, A 0.000, B 0.000, C 0.000 }
gfCNCPoint1[21592] = {X 195.3825, Y 56.9774, Z -2.1667, A 0.000, B 0.000, C 0.000 }
gfCNCPoint1[21593] = {X 199.6722, Y 61.6591, Z -2.1667, A 0.000, B 0.000, C 0.000 }
gfCNCPoint1[21594] = {X 202.0407, Y 61.2716, Z -2.1667, A 0.000, B 0.000, C 0.000 }
gfCNCPoint1[21595] = {X 201.9014, Y 60.1432, Z -2.1667, A 0.000, B 0.000, C 0.000 }
gfCNCPoint1[21596] = {X 201.8510, Y 59.0073, Z -2.1667, A 0.000, B 0.000, C 0.000 }
gfCNCPoint1[21597] = {X 201.8508, Y 58.0000, Z -2.1667, A 0.000, B 0.000, C 0.000 }
gfCNCPoint1[21598] = {X 201.9283, Y 56.5036, Z -2.1667, A 0.000, B 0.000, C 0.000 }
gfCNCPoint1[21599] = {X 202.1601, Y 55.0232, Z -2.1667, A 0.000, B 0.000, C 0.000 }
gfCNCPoint1[21600] = {X 202.4970, Y 53.7228, Z -2.1667, A 0.000, B 0.000, C 0.000 }
gfCNCPoint1[21601] = {X 202.9529, Y 52.4591, Z -2.1667, A 0.000, B 0.000, C 0.000 }
gfCNCPoint1[21602] = {X 203.5239, Y 51.2432, Z -2.1667, A 0.000, B 0.000, C 0.000 }
gfCNCPoint1[21603] = {X 202.2642, Y 51.6547, Z -2.1667, A 0.000, B 0.000, C 0.000 }
gfCNCPoint1[21604] = {X 200.9602, Y 51.8905, Z -2.1667, A 0.000, B 0.000, C 0.000 }
gfCNCPoint1[21605] = {X 199.6362, Y 51.9463, Z -2.1667, A 0.000, B 0.000, C 0.000 }
gfCNCPoint1[21606] = {X 199.2152, Y 52.1547, Z -2.1667, A 0.000, B 0.000, C 0.000 }
gfCNCPoint1[21607] = {X 198.7914, Y 52.3573, Z -2.1667, A 0.000, B 0.000, C 0.000 }
gfCNCPoint1[21608] = {X 196.7763, Y 53.2251, Z -2.1667, A 0.000, B 0.000, C 0.000 }
gfCNCPoint1[21609] = {X 194.7095, Y 53.9611, Z -2.1667, A 0.000, B 0.000, C 0.000 }
gfCNCPoint1[21610] = {X 192.5995, Y 54.5623, Z -2.1667, A 0.000, B 0.000, C 0.000 }
gfCNCPoint1[21611] = {X 192.9063, Y 56.2412, Z -2.1667, A 0.000, B 0.000, C 0.000 }
gfCNCPoint1[21612] = {X 193.0134, Y 57.9444, Z -2.1667, A 0.000, B 0.000, C 0.000 }
gfCNCPoint1[21613] = {X 210.3938, Y 76.9129, Z -2.1667, A 0.000, B 0.000, C 0.000 }
gfCNCPoint1[21614] = {X 208.6243, Y 78.5343, Z -2.1667, A 0.000, B 0.000, C 0.000 }
gfCNCPoint1[21615] = {X 214.3884, Y 84.8250, Z -2.1667, A 0.000, B 0.000, C 0.000 }
gfCNCPoint1[21616] = {X 228.8383, Y 75.5676, Z -2.1667, A 0.000, B 0.000, C 0.000 }
gfCNCPoint1[21617] = {X 218.7728, Y 71.6174, Z -2.1667, A 0.000, B 0.000, C 0.000 }
gfCNCPoint1[21618] = {X 217.8436, Y 71.3038, Z -2.1667, A 0.000, B 0.000, C 0.000 }
